# B&R Automation Studio project TD52 (part 48)

```iecst
	xMsg2303();

	OUT_CU.bMsg2303 :=	xMsg2303.Q;
	MM2VIS.bMsg2303 :=	xMsg2303.Q;

	(* W2415 mains import controller: Messsignalstörung Netzbezugs- Sollwert 	*)
	xMsg2415.Enable := bMsg2415_Enable AND IN_CU.tPB2MM.bParaSetupOk;
	xMsg2415.Set 	:= bMsg2415_Set;
	xMsg2415.PT 	:= T#1s;
	xMsg2415.Prio 	:= 4;
	xMsg2415.Reset 	:= FALSE;

	xMsg2415();

	OUT_CU.bMsg2415 :=	xMsg2415.Q;
	MM2VIS.bMsg2415 :=	xMsg2415.Q;

	(* W2416 mains import controller: Messsignalstörung Netzbezugs- Istwert	*)
//	Para.bP_Mns_AnaIn_Enable := NOT Para.bP_Mns_MMU_Enable	;						(*necessary, because bP_Mns_AnaIn_Enable is not a parameter on VIS anymore*)

	xMsg2416.Enable := bMsg2416_Enable AND IN_CU.tPB2MM.bParaSetupOk;
	xMsg2416.Set 	:= bMsg2416_Set;
//	NOT IN_CU.tP_Mns_AnaIn.GoodQual;
	xMsg2416.PT		:= T#1s;
	xMsg2416.Prio 	:= 4;
	xMsg2416.Reset 	:= FALSE;

	xMsg2416();

	OUT_CU.bMsg2416 :=	xMsg2416.Q;
	MM2VIS.bMsg2416 :=	xMsg2416.Q;

	(* W2417 mains export power limit: Warning, if NEGATIVE Mains Import (= power export to the grid) is exceeding (<) the allowed limit (-Limit value)  *)
	xMsg2417.Enable := bMsg2417_Enable AND IN_CU.tPB2MM.bParaSetupOk;
	xMsg2417.Set 	:= bMsg2417_Set;
	xMsg2417.PT 	:= T#1s;
	xMsg2417.Prio 	:= 4;
	xMsg2417.Reset 	:= FALSE;
	xMsg2417();

	OUT_CU.bMsg2417 :=	xMsg2417.Q;
	MM2VIS.bMsg2417 :=	xMsg2417.Q;

	(* W2418  mains import controller limit 2:  Warning if positive Mains Import (= power drawn from the grid) is exceeding (>) the allowed limit (+Limit value)*)
	xMsg2418.Enable := bMsg2418_Enable AND IN_CU.tPB2MM.bParaSetupOk;
	xMsg2418.Set 	:= bMsg2418_Set;
	xMsg2418.PT 	:= T#1s;
	xMsg2418.Prio 	:= 4;
	xMsg2418.Reset 	:= FALSE;

	xMsg2418();

	OUT_CU.bMsg2418 :=	xMsg2418.Q;
	MM2VIS.bMsg2418 :=	xMsg2418.Q;

	(* B2419 operating message mns import ctr: Engine Demand Off (ex.Warning W2419) *)
	TP_EngDSS_Mains_Off(IN := NOT(OUT_CU.bEngDSS_Mains), PT := T#11s);
	xMsg2419.Enable := 	Para.bCtr_Mns_Enable;
	xMsg2419.Set := 	TP_EngDSS_Mains_Off.Q;
	xMsg2419.PT := 		T#1s;
	xMsg2419.Prio := 	5;
	IF xMsg2419.Set THEN iReset_Msg2419 := iDelay_MsgAutoReset_100ms; ELSE iReset_Msg2419 := LIMIT(0, iReset_Msg2419 -1,32767); END_IF		(* activate 'Message Hold Time' to avoid log clathering by repeated OpMsg entries *)
	xMsg2419.Reset := 	iReset_Msg2419 < 1;		//.Reset := TRUE;
//
	xMsg2419();
//
	OUT_CU.bMsg2419 :=		xMsg2419.Q;	//  := TP_EngDSS_Mains_Off.Q;	//
	MM2VIS.bMsg2419 :=		xMsg2419.Q;	//	:= TP_EngDSS_Mains_Off.Q;	//

	(* B2420 operating message mns import ctr: Engine Demand On (ex. warning W2420)*)
	TP_EngDSS_Mains(IN := OUT_CU.bEngDSS_Mains, PT := T#11s);
	xMsg2420.Enable := 	Para.bCtr_Mns_Enable;
	xMsg2420.Set := 	TP_EngDSS_Mains.Q;
	xMsg2420.PT := 		T#1s;
	xMsg2420.Prio := 	5;

	IF xMsg2420.Set THEN iReset_Msg2420 := iDelay_MsgAutoReset_100ms; ELSE iReset_Msg2420 := LIMIT(0, iReset_Msg2420 -1,32767); END_IF		(* activate 'Message Hold Time' to avoid log clathering by repeated OpMsg entries *)
	xMsg2420.Reset := 	iReset_Msg2420 < 1;		//.Reset := TRUE;
//
	xMsg2420();
//
	OUT_CU.bMsg2420 :=		xMsg2420.Q;		// := TP_EngDSS_Mains.Q;		//
	MM2VIS.bMsg2420 :=		xMsg2420.Q;		// := TP_EngDSS_Mains.Q;		//

(*  Debug Info only (may be removed in tested versions)  *)
	bCtr_Mns_Options_2	:= Para.iCtr_Mns_Options.2;
	bCtr_Mns_Options_3	:= Para.iCtr_Mns_Options.3;
	bCtr_Mns_Options_4	:= Para.iCtr_Mns_Options.4;
	bCtr_Mns_Options_5	:= Para.iCtr_Mns_Options.5;
	bCtr_Mns_Options_6	:= Para.iCtr_Mns_Options.6;
	bCtr_Mns_Options_7	:= Para.iCtr_Mns_Options.7;
	bCtr_Mns_Options_8	:= Para.iCtr_Mns_Options.8;			bCtr_Mns_Options_1;	bCtr_Mns_Options_9;	bCtr_Mns_Options_0;
	R_TRIG_Options(CLK := (VIS2MM.tCtr_Mns_In.Tune_PI OR VIS2MM.tCtr_Mns_In.Tune_PID) AND VIS2MM.tCtr_Mns_In.Tune_quality>0);
	IF R_TRIG_Options.Q AND IN_CU.iIdx_OMSS=0 THEN Para.iCtr_Mns_Options := Para.iCtr_Mns_Options + BOOL_TO_INT(VIS2MM.tCtr_Mns_In.Tune_PI) * VIS2MM.tCtr_Mns_In.Tune_quality - BOOL_TO_INT(VIS2MM.tCtr_Mns_In.Tune_PID) * VIS2MM.tCtr_Mns_In.Tune_quality ; END_IF			(*Debug options*)

	(*********************************************************)

		(* W3565 Messsignalstörung Generator Leistungssollwert *)
		xMsg3565.Enable := 	(Para.rI_P_Set_ExtAI_NormScalMin >= 0.004);  (* if signal check is ok AND scaling parameter Min has to be set >4mA*) 	(*old V3.40: monitoring active, if parameter p_soll_i1 is setted to 4mA or higher *)
		xMsg3565.Set := 	NOT IN_CU.tP_Set_ExtAI_Norm.GoodQual;
		xMsg3565.PT := 		T#2s;
		xMsg3565.Prio := 	4;
		xMsg3565.Reset := 	FALSE;

		xMsg3565();

		MM2VIS.bMsg3565 :=	xMsg3565.Q;
		OUT_CU.bMsg3565 :=	xMsg3565.Q;

		(* W9285 Measuring signal failure external voltage setpoint *)
		MM2VIS.bMsg9285 :=	IN_CU.bMsg[9285];

		(* W9286 Measuring signal failure external speed setpoint (Isolated operation) *)
		xMsg9286.Enable := 	(Para.rI_N_Set_ExtAI_NormScalMin >= 0.004) AND IN_CU.tN_Set_ExtAI_Norm.Exist AND IN_CU.tPB2MM.bParaSetupOk;
		xMsg9286.Set := 	NOT IN_CU.tN_Set_ExtAI_Norm.GoodQual;
		xMsg9286.PT := 		T#1s;
		xMsg9286.Prio := 	4;
		xMsg9286.Reset := 	FALSE;

		xMsg9286();

		MM2VIS.bMsg9286 :=	xMsg9286.Q;
		OUT_CU.bMsg9286 :=	xMsg9286.Q;

		(* W9287 Failure external speed / voltage controller *)
		xMsg9287.Enable := 	IN_CU.tExtCtrOk.GoodQual AND IN_CU.tPB2MM.bParaSetupOk;
		xMsg9287.Set := 	NOT IN_CU.tExtCtrOk.Di;
		xMsg9287.PT := 		T#1s;
		xMsg9287.Prio := 	4;
		xMsg9287.Reset := 	FALSE;

		xMsg9287();

		MM2VIS.bMsg9287 :=	xMsg9287.Q;
		OUT_CU.bMsg9287 :=	xMsg9287.Q;

	(*----------------------------------------------------------------------------*)
	(* OPERATING MESSAGES: connect activation bits here customized 				  *)
	(*----------------------------------------------------------------------------*)

		OUT_CU.bMsg3232;// :=		FALSE;	(* B3232 reserve operating message 1 *)
		OUT_CU.bMsg3233;// :=		FALSE;	(* B3233 reserve operating message 2 *)
		OUT_CU.bMsg3234 ;// :=		FALSE;	(* B3234 reserve operating message 3 *)
		OUT_CU.bMsg3235 ;// :=		FALSE;	(* B3235 reserve operating message 4 *)
		OUT_CU.bMsg3236 ;// := 		FALSE;	(* B3236 reserve operating message 5 *)
		OUT_CU.bMsg3237 ;// := 		FALSE;	(* B3237 reserve operating message 6 *)

		OUT_CU.bMsg3250 ;// := 		FALSE;	(* B3250 reserve operating message 7 *)
		OUT_CU.bMsg3251 ;// := 		FALSE;	(* B3251 reserve operating message 8 *)

		OUT_CU.bMsg3601 ;// := 		FALSE;	(* B3601 reserve operating message 9 *)
		OUT_CU.bMsg3602 ;// := 		FALSE;	(* B3602 reserve operating message 10 *)
		OUT_CU.bMsg3603 ;// := 		FALSE;	(* B3603 reserve operating message 11 *)
		OUT_CU.bMsg3604 ;// := 		FALSE;	(* B3604 reserve operating message 12 *)
		OUT_CU.bMsg3605 ;// := 		FALSE;	(* B3605 reserve operating message 13 *)
		OUT_CU.bMsg3606 ;// := 		FALSE;	(* B3606 reserve operating message 14 *)
		OUT_CU.bMsg3607 ;// := 		FALSE;	(* B3607 reserve operating message 15 *)
		OUT_CU.bMsg3608 ;// := 		FALSE;	(* B3608 reserve operating message 16 *)
		OUT_CU.bMsg3609 ;// := 		FALSE;	(* B3609 reserve operating message 17 *)
		OUT_CU.bMsg3610 ;// := 		FALSE;	(* B3610 reserve operating message 18 *)

		OUT_CU.bMsg3611 ;// := 		FALSE;	(* B3611 reserve operating message 19 *)
		OUT_CU.bMsg3612 ;// := 		FALSE;	(*  	 reserve operating message 20 *)
		OUT_CU.bMsg3613 ;// := 		FALSE;	(* 		 reserve operating message 21 *)
		OUT_CU.bMsg3614 ;// := 		FALSE;	(* 		 reserve operating message 22 *)
		OUT_CU.bMsg3615 ;// := 		FALSE;	(* 		 reserve operating message 23 *)
		OUT_CU.bMsg3616 ;// := 		FALSE;	(* 		 reserve operating message 24 *)
		OUT_CU.bMsg3617 ;// := 		FALSE;	(* 		 reserve operating message 25 *)
		OUT_CU.bMsg3618 ;// := 		FALSE;	(* 		 reserve operating message 26 *)
		OUT_CU.bMsg3619 ;// := 		FALSE;	(* 		 reserve operating message 27 *)
		OUT_CU.bMsg3620 ;// := 		FALSE;	(* 		 reserve operating message 28 *)

		OUT_CU.bMsg3621 ;// := 		FALSE;	(* B3621 reserve operating message 29 *)
		OUT_CU.bMsg3622 ;// := 		FALSE;	(* 		 reserve operating message 30 *)
		OUT_CU.bMsg3623 ;// := 		FALSE;	(* 		 reserve operating message 31 *)
		OUT_CU.bMsg3624 ;// := 		FALSE;	(* 		 reserve operating message 32 *)
		OUT_CU.bMsg3625 ;// := 		FALSE;	(* 		 reserve operating message 33 *)
		OUT_CU.bMsg3626 ;// := 		FALSE;	(* 		 reserve operating message 34 *)
		OUT_CU.bMsg3627 ;// := 		FALSE;	(* 		 reserve operating message 35 *)
		OUT_CU.bMsg3628 ;// := 		FALSE;	(* 		 reserve operating message 36 *)
		OUT_CU.bMsg3629 ;// := 		FALSE;	(* 		 reserve operating message 37 *)
		OUT_CU.bMsg3630 ;// := 		FALSE;	(* 		 reserve operating message 38 *)

		OUT_CU.bMsg3631 ;// := 		FALSE;	(* 		 reserve operating message 39 *)
		OUT_CU.bMsg3632 ;// := 		FALSE;	(* 		 reserve operating message 40 *)
		OUT_CU.bMsg3633 ;// := 		FALSE;	(* 		 reserve operating message 41 *)
		OUT_CU.bMsg3634 ;// := 		FALSE;	(* 		 reserve operating message 42 *)
		OUT_CU.bMsg3635 ;// := 		FALSE;	(* 		 reserve operating message 43 *)
		OUT_CU.bMsg3636 ;// := 		FALSE;	(* 		 reserve operating message 44 *)
		OUT_CU.bMsg3637 ;// := 		FALSE;	(* 		 reserve operating message 45 *)
		OUT_CU.bMsg3638 ;// := 		FALSE;	(* 		 reserve operating message 46 *)
		OUT_CU.bMsg3639 ;// := 		FALSE;	(* 		 reserve operating message 47 *)
		OUT_CU.bMsg3640 ;// := 		FALSE;	(* 		 reserve operating message 48 *)

		OUT_CU.bMsg3641 ;// := 		FALSE;	(* B3641 reserve operating message 49 *)
		OUT_CU.bMsg3642 ;// := 		FALSE;	(* 		 reserve operating message 50 *)
		OUT_CU.bMsg3643 ;// := 		FALSE;	(* 		 reserve operating message 51 *)
		OUT_CU.bMsg3644 ;// := 		FALSE;	(* 		 reserve operating message 52 *)
		OUT_CU.bMsg3645 ;// := 		FALSE;	(* 		 reserve operating message 53 *)
		OUT_CU.bMsg3646 ;// := 		FALSE;	(* 		 reserve operating message 54 *)
		OUT_CU.bMsg3647 ;// := 		FALSE;	(* 		 reserve operating message 55 *)
		OUT_CU.bMsg3648 ;// := 		FALSE;	(* 		 reserve operating message 56 *)
		OUT_CU.bMsg3649 ;// := 		FALSE;	(* 		 reserve operating message 57 *)
		OUT_CU.bMsg3650 ;// := 		FALSE;	(* 		 reserve operating message 58 *)

		OUT_CU.bMsg3651 ;// := 		FALSE;	(* 		 reserve operating message 59 *)
		OUT_CU.bMsg3652 ;// := 		FALSE;	(* 		 reserve operating message 60 *)
		OUT_CU.bMsg3653 ;// := 		FALSE;	(* 		 reserve operating message 61 *)
		OUT_CU.bMsg3654 ;// := 		FALSE;	(* 		 reserve operating message 62 *)
		OUT_CU.bMsg3655 ;// := 		FALSE;	(* 		 reserve operating message 63 *)
		OUT_CU.bMsg3656 ;// := 		FALSE;	(* 		 reserve operating message 64 *)
		OUT_CU.bMsg3657 ;// := 		FALSE;	(* 		 reserve operating message 65 *)
		OUT_CU.bMsg3658 ;// := 		FALSE;	(* 		 reserve operating message 66 *)
		OUT_CU.bMsg3659 ;// := 		FALSE;	(* 		 reserve operating message 67 *)
		OUT_CU.bMsg3660 ;// := 		FALSE;	(* 		 reserve operating message 68 *)

		OUT_CU.bMsg3661 ;// := 		FALSE;	(* B3661 reserve operating message 69 *)
		OUT_CU.bMsg3662 ;// := 		FALSE;	(* 		 reserve operating message 70 *)
		OUT_CU.bMsg3663 ;// := 		FALSE;	(* 		 reserve operating message 71 *)
		OUT_CU.bMsg3664 ;// := 		FALSE;	(* 		 reserve operating message 72 *)
		OUT_CU.bMsg3665 ;// := 		FALSE;	(* 		 reserve operating message 73 *)
		OUT_CU.bMsg3666 ;// := 		FALSE;	(* 		 reserve operating message 74 *)
		OUT_CU.bMsg3667 ;// := 		FALSE;	(* 		 reserve operating message 75 *)
		OUT_CU.bMsg3668 ;// := 		FALSE;	(* 		 reserve operating message 76 *)
		OUT_CU.bMsg3669 ;// := 		FALSE;	(* 		 reserve operating message 77 *)
		OUT_CU.bMsg3670 ;// := 		FALSE;	(* 		 reserve operating message 78 *)

		OUT_CU.bMsg3671 ;// := 		FALSE;	(* 		 reserve operating message 79 *)
		OUT_CU.bMsg3672 ;// := 		FALSE;	(* 		 reserve operating message 80 *)
		OUT_CU.bMsg3673 ;// := 		FALSE;	(* 		 reserve operating message 81 *)
		OUT_CU.bMsg3674 ;// := 		FALSE;	(* 		 reserve operating message 82 *)
		OUT_CU.bMsg3675 ;// := 		FALSE;	(* 		 reserve operating message 83 *)
		OUT_CU.bMsg3676 ;// := 		FALSE;	(* 		 reserve operating message 84 *)
		OUT_CU.bMsg3677 ;// := 		FALSE;	(* 		 reserve operating message 85 *)
		OUT_CU.bMsg3678 ;// := 		FALSE;	(* 		 reserve operating message 86 *)
		OUT_CU.bMsg3679 ;// := 		FALSE;	(* 		 reserve operating message 87 *)
		OUT_CU.bMsg3680 ;// := 		FALSE;	(* 		 reserve operating message 88 *)

		OUT_CU.bMsg3681 ;// := 		FALSE;	(* B3681 reserve operating message 89 *)
		OUT_CU.bMsg3682 ;// := 		FALSE;	(* 		 reserve operating message 90 *)
		OUT_CU.bMsg3683 ;// := 		FALSE;	(* 		 reserve operating message 91 *)
		OUT_CU.bMsg3684 ;// := 		FALSE;	(* 		 reserve operating message 92 *)
		OUT_CU.bMsg3685 ;// := 		FALSE;	(* 		 reserve operating message 93 *)
		OUT_CU.bMsg3686 ;// := 		FALSE;	(* 		 reserve operating message 94 *)
		OUT_CU.bMsg3687 ;// := 		FALSE;	(* 		 reserve operating message 95 *)
		OUT_CU.bMsg3688 ;// := 		FALSE;	(* 		 reserve operating message 96 *)
		OUT_CU.bMsg3689 ;// := 		FALSE;	(* 		 reserve operating message 97 *)
		OUT_CU.bMsg3690 ;// := 		FALSE;	(* 		 reserve operating message 98 *)

		OUT_CU.bMsg3691 ;// := 		FALSE;	(* 		 reserve operating message 99 *)
		OUT_CU.bMsg3692 ;// := 		FALSE;	(* 		 reserve operating message 100 *)
		OUT_CU.bMsg3693 ;// := 		FALSE;	(* 		 reserve operating message 101 *)
		OUT_CU.bMsg3694 ;// := 		FALSE;	(* 		 reserve operating message 102 *)
		OUT_CU.bMsg3695 ;// := 		FALSE;	(* 		 reserve operating message 103 *)
		OUT_CU.bMsg3696 ;// := 		FALSE;	(* 		 reserve operating message 104 *)
		OUT_CU.bMsg3697 ;// := 		FALSE;	(* 		 reserve operating message 105 *)
		OUT_CU.bMsg3698 ;// := 		FALSE;	(* 		 reserve operating message 106 *)
		OUT_CU.bMsg3699 ;// := 		FALSE;	(* 		 reserve operating message 107 *)
		OUT_CU.bMsg3700 ;// := 		FALSE;	(* 		 reserve operating message 108 *)

		OUT_CU.bMsg6701 ;// := 		FALSE;	(* B6701 reserve operating message 109 *) (*import HMI Extension *)
		OUT_CU.bMsg6702 ;// := 		FALSE;	(* B6702 reserve operating message 110 *) (*import HMI Extension *)
		OUT_CU.bMsg6703 ;// := 		FALSE;	(* B6703 reserve operating message 111 *) (*import HMI Extension *)
		OUT_CU.bMsg6704 ;// := 		FALSE;	(* B6704 reserve operating message 112 *) (*import HMI Extension *)
		OUT_CU.bMsg6705 ;// := 		FALSE;	(* B6705 reserve operating message 113 *) (*import HMI Extension *)
		OUT_CU.bMsg6706 ;// := 		FALSE;	(* B6706 reserve operating message 114 *) (*import HMI Extension *)
		OUT_CU.bMsg6707 ;// := 		FALSE;	(* B6707 reserve operating message 115 *) (*import HMI Extension *)
		OUT_CU.bMsg6708 ;// := 		FALSE;	(* B6708 reserve operating message 116 *) (*import HMI Extension *)
		OUT_CU.bMsg6709 ;// := 		FALSE;	(* B6709 reserve operating message 117 *) (*import HMI Extension *)
		OUT_CU.bMsg6710 ;// := 		FALSE;	(* B6710 reserve operating message 118 *) (*import HMI Extension *)

		OUT_CU.bMsg6711 ;// := 		FALSE;	(* B6711 reserve operating message 119 *) (*import HMI Extension *)
		OUT_CU.bMsg6712 ;// := 		FALSE;	(* B6712 reserve operating message 120 *) (*import HMI Extension *)
		OUT_CU.bMsg6713 ;// := 		FALSE;	(* B6713 reserve operating message 121 *) (*import HMI Extension *)
		OUT_CU.bMsg6714 ;// := 		FALSE;	(* B6714 reserve operating message 122 *) (*import HMI Extension *)
		OUT_CU.bMsg6715 ;// := 		FALSE;	(* B6715 reserve operating message 123 *) (*import HMI Extension *)
		OUT_CU.bMsg6716 ;// := 		FALSE;	(* B6716 reserve operating message 124 *) (*import HMI Extension *)
		OUT_CU.bMsg6717 ;// := 		FALSE;	(* B6717 reserve operating message 125 *) (*import HMI Extension *)
		OUT_CU.bMsg6718 ;// := 		FALSE;	(* B6718 reserve operating message 126 *) (*import HMI Extension *)
		OUT_CU.bMsg6719 ;// := 		FALSE;	(* B6719 reserve operating message 127 *) (*import HMI Extension *)
		OUT_CU.bMsg6720 ;// := 		FALSE;	(* B6720 reserve operating message 128 *) (*import HMI Extension *)

		OUT_CU.bMsg6721 ;// := 		FALSE;	(* B6721 reserve operating message 129 *) (*import HMI Extension *)
		OUT_CU.bMsg6722 ;// := 		FALSE;	(* B6722 reserve operating message 130 *) (*import HMI Extension *)
		OUT_CU.bMsg6723 ;// := 		FALSE;	(* B6723 reserve operating message 131 *) (*import HMI Extension *)
		OUT_CU.bMsg6724 ;// := 		FALSE;	(* B6724 reserve operating message 132 *) (*import HMI Extension *)
		OUT_CU.bMsg6725 ;// := 		FALSE;	(* B6725 reserve operating message 133 *) (*import HMI Extension *)
		OUT_CU.bMsg6726 ;// := 		FALSE;	(* B6726 reserve operating message 134 *) (*import HMI Extension *)
		OUT_CU.bMsg6727 ;// := 		FALSE;	(* B6727 reserve operating message 135 *) (*import HMI Extension *)
		OUT_CU.bMsg6728 ;// := 		FALSE;	(* B6728 reserve operating message 136 *) (*import HMI Extension *)
		OUT_CU.bMsg6729 ;// := 		FALSE;	(* B6729 reserve operating message 137 *) (*import HMI Extension *)
		OUT_CU.bMsg6730 ;// := 		FALSE;	(* B6730 reserve operating message 138 *) (*import HMI Extension *)

		OUT_CU.bMsg6731 ;// := 		FALSE;	(* B6731 reserve operating message 139 *) (*import HMI Extension *)
		OUT_CU.bMsg6732 ;// := 		FALSE;	(* B6732 reserve operating message 140 *) (*import HMI Extension *)
		OUT_CU.bMsg6733 ;// := 		FALSE;	(* B6733 reserve operating message 141 *) (*import HMI Extension *)
		OUT_CU.bMsg6734 ;// := 		FALSE;	(* B6734 reserve operating message 142 *) (*import HMI Extension *)
		OUT_CU.bMsg6735 ;// := 		FALSE;	(* B6735 reserve operating message 143 *) (*import HMI Extension *)
		OUT_CU.bMsg6736 ;// := 		FALSE;	(* B6736 reserve operating message 144 *) (*import HMI Extension *)
		OUT_CU.bMsg6737 ;// := 		FALSE;	(* B6737 reserve operating message 145 *) (*import HMI Extension *)
		OUT_CU.bMsg6738 ;// := 		FALSE;	(* B6738 reserve operating message 146 *) (*import HMI Extension *)
		OUT_CU.bMsg6739 ;// := 		FALSE;	(* B6739 reserve operating message 147 *) (*import HMI Extension *)
		OUT_CU.bMsg6740 ;// := 		FALSE;	(* B6740 reserve operating message 148 *) (*import HMI Extension *)

		OUT_CU.bMsg6741 ;// := 		FALSE;	(* B6741 reserve operating message 149 *) (*import HMI Extension *)
		OUT_CU.bMsg6742 ;// := 		FALSE;	(* B6742 reserve operating message 150 *) (*import HMI Extension *)
		OUT_CU.bMsg6743 ;// := 		FALSE;	(* B6743 reserve operating message 151 *) (*import HMI Extension *)
		OUT_CU.bMsg6744 ;// := 		FALSE;	(* B6744 reserve operating message 152 *) (*import HMI Extension *)
		OUT_CU.bMsg6745 ;// := 		FALSE;	(* B6745 reserve operating message 153 *) (*import HMI Extension *)
		OUT_CU.bMsg6746 ;// := 		FALSE;	(* B6746 reserve operating message 154 *) (*import HMI Extension *)
		OUT_CU.bMsg6747 ;// := 		FALSE;	(* B6747 reserve operating message 155 *) (*import HMI Extension *)
		OUT_CU.bMsg6748 ;// := 		FALSE;	(* B6748 reserve operating message 156 *) (*import HMI Extension *)
		OUT_CU.bMsg6749 ;// := 		FALSE;	(* B6749 reserve operating message 157 *) (*import HMI Extension *)
		OUT_CU.bMsg6750 ;// := 		FALSE;	(* B6750 reserve operating message 158 *) (*import HMI Extension *)

		OUT_CU.bMsg6751 ;// := 		FALSE;	(* B6751 reserve operating message 159 *) (*import HMI Extension *)
		OUT_CU.bMsg6752 ;// := 		FALSE;	(* B6752 reserve operating message 160 *) (*import HMI Extension *)
		OUT_CU.bMsg6753 ;// := 		FALSE;	(* B6753 reserve operating message 161 *) (*import HMI Extension *)
		OUT_CU.bMsg6754 ;// := 		FALSE;	(* B6754 reserve operating message 162 *) (*import HMI Extension *)
		OUT_CU.bMsg6755 ;// := 		FALSE;	(* B6755 reserve operating message 163 *) (*import HMI Extension *)
		OUT_CU.bMsg6756 ;// := 		FALSE;	(* B6756 reserve operating message 164 *) (*import HMI Extension *)
		OUT_CU.bMsg6757 ;// := 		FALSE;	(* B6757 reserve operating message 165 *) (*import HMI Extension *)
		OUT_CU.bMsg6758 ;// := 		FALSE;	(* B6758 reserve operating message 166 *) (*import HMI Extension *)
		OUT_CU.bMsg6759 ;// := 		FALSE;	(* B6759 reserve operating message 167 *) (*import HMI Extension *)
		OUT_CU.bMsg6760 ;// := 		FALSE;	(* B6760 reserve operating message 168 *) (*import HMI Extension *)

		OUT_CU.bMsg6761 ;// := 		FALSE;	(* B6761 reserve operating message 169 *) (*import HMI Extension *)
		OUT_CU.bMsg6762 ;// := 		FALSE;	(* B6762 reserve operating message 170 *) (*import HMI Extension *)
		OUT_CU.bMsg6763 ;// := 		FALSE;	(* B6763 reserve operating message 171 *) (*import HMI Extension *)
		OUT_CU.bMsg6764 ;// := 		FALSE;	(* B6764 reserve operating message 172 *) (*import HMI Extension *)
		OUT_CU.bMsg6765 ;// := 		FALSE;	(* B6765 reserve operating message 173 *) (*import HMI Extension *)
		OUT_CU.bMsg6766 ;// := 		FALSE;	(* B6766 reserve operating message 174 *) (*import HMI Extension *)
		OUT_CU.bMsg6767 ;// := 		FALSE;	(* B6767 reserve operating message 175 *) (*import HMI Extension *)
		OUT_CU.bMsg6768 ;// := 		FALSE;	(* B6768 reserve operating message 176 *) (*import HMI Extension *)
		OUT_CU.bMsg6769 ;// := 		FALSE;	(* B6769 reserve operating message 177 *) (*import HMI Extension *)
		OUT_CU.bMsg6770 ;// := 		FALSE;	(* B6770 reserve operating message 178 *) (*import HMI Extension *)

		OUT_CU.bMsg6771 ;// := 		FALSE;	(* B6771 reserve operating message 179 *) (*import HMI Extension *)
		OUT_CU.bMsg6772 ;// := 		FALSE;	(* B6772 reserve operating message 180 *) (*import HMI Extension *)
		OUT_CU.bMsg6773 ;// := 		FALSE;	(* B6773 reserve operating message 181 *) (*import HMI Extension *)
		OUT_CU.bMsg6774 ;// := 		FALSE;	(* B6774 reserve operating message 182 *) (*import HMI Extension *)
		OUT_CU.bMsg6775 ;// := 		FALSE;	(* B6775 reserve operating message 183 *) (*import HMI Extension *)
		OUT_CU.bMsg6776 ;// := 		FALSE;	(* B6776 reserve operating message 184 *) (*import HMI Extension *)
		OUT_CU.bMsg6777 ;// := 		FALSE;	(* B6777 reserve operating message 185 *) (*import HMI Extension *)
		OUT_CU.bMsg6778 ;// := 		FALSE;	(* B6778 reserve operating message 186 *) (*import HMI Extension *)
		OUT_CU.bMsg6779 ;// := 		FALSE;	(* B6779 reserve operating message 187 *) (*import HMI Extension *)
		OUT_CU.bMsg6780 ;// := 		FALSE;	(* B6780 reserve operating message 188 *) (*import HMI Extension *)

		OUT_CU.bMsg6781 ;// := 		FALSE;	(* B6781 reserve operating message 189 *) (*import HMI Extension *)
		OUT_CU.bMsg6782 ;// := 		FALSE;	(* B6782 reserve operating message 190 *) (*import HMI Extension *)
		OUT_CU.bMsg6783 ;// := 		FALSE;	(* B6783 reserve operating message 191 *) (*import HMI Extension *)
		OUT_CU.bMsg6784 ;// := 		FALSE;	(* B6784 reserve operating message 192 *) (*import HMI Extension *)
		OUT_CU.bMsg6785 ;// := 		FALSE;	(* B6785 reserve operating message 193 *) (*import HMI Extension *)
		OUT_CU.bMsg6786 ;// := 		FALSE;	(* B6786 reserve operating message 194 *) (*import HMI Extension *)
		OUT_CU.bMsg6787 ;// := 		FALSE;	(* B6787 reserve operating message 195 *) (*import HMI Extension *)
		OUT_CU.bMsg6788 ;// := 		FALSE;	(* B6788 reserve operating message 196 *) (*import HMI Extension *)
		OUT_CU.bMsg6789 ;// := 		FALSE;	(* B6789 reserve operating message 197 *) (*import HMI Extension *)
		OUT_CU.bMsg6790 ;// := 		FALSE;	(* B6790 reserve operating message 198 *) (*import HMI Extension *)

		OUT_CU.bMsg6791 ;// := 		FALSE;	(* B6791 reserve operating message 199 *) (*import HMI Extension *)
		OUT_CU.bMsg6792 ;// := 		FALSE;	(* B6792 reserve operating message 200 *) (*import HMI Extension *)
		OUT_CU.bMsg6793 ;// := 		FALSE;	(* B6793 reserve operating message 201 *) (*import HMI Extension *)
		OUT_CU.bMsg6794 ;// := 		FALSE;	(* B6794 reserve operating message 202 *) (*import HMI Extension *)
		OUT_CU.bMsg6795 ;// := 		FALSE;	(* B6795 reserve operating message 203 *) (*import HMI Extension *)
		OUT_CU.bMsg6796 ;// := 		FALSE;	(* B6796 reserve operating message 204 *) (*import HMI Extension *)
		OUT_CU.bMsg6797 ;// := 		FALSE;	(* B6797 reserve operating message 205 *) (*import HMI Extension *)
		OUT_CU.bMsg6798 ;// := 		FALSE;	(* B6798 reserve operating message 206 *) (*import HMI Extension *)
		OUT_CU.bMsg6799 ;// := 		FALSE;	(* B6799 reserve operating message 207 *) (*import HMI Extension *)
		OUT_CU.bMsg6800 ;// := 		FALSE;	(* B6800 reserve operating message 208 *) (*import HMI Extension *)

		OUT_CU.bMsg6801 ;// := 		FALSE;	(* B6801 reserve operating message 209 *) (*import HMI Extension *)
		OUT_CU.bMsg6802 ;// := 		FALSE;	(* B6802 reserve operating message 210 *) (*import HMI Extension *)
		OUT_CU.bMsg6803 ;// := 		FALSE;	(* B6803 reserve operating message 211 *) (*import HMI Extension *)
		OUT_CU.bMsg6804 ;// := 		FALSE;	(* B6804 reserve operating message 212 *) (*import HMI Extension *)
		OUT_CU.bMsg6805 ;// := 		FALSE;	(* B6805 reserve operating message 213 *) (*import HMI Extension *)
		OUT_CU.bMsg6806 ;// := 		FALSE;	(* B6806 reserve operating message 214 *) (*import HMI Extension *)
		OUT_CU.bMsg6807 ;// := 		FALSE;	(* B6807 reserve operating message 215 *) (*import HMI Extension *)
		OUT_CU.bMsg6808 ;// := 		FALSE;	(* B6808 reserve operating message 216 *) (*import HMI Extension *)
		OUT_CU.bMsg6809 ;// := 		FALSE;	(* B6809 reserve operating message 217 *) (*import HMI Extension *)
		OUT_CU.bMsg6810 ;// := 		FALSE;	(* B6810 reserve operating message 218 *) (*import HMI Extension *)

		OUT_CU.bMsg6811 ;// := 		FALSE;	(* B6811 reserve operating message 219 *) (*import HMI Extension *)
		OUT_CU.bMsg6812 ;// := 		FALSE;	(* B6812 reserve operating message 220 *) (*import HMI Extension *)
		OUT_CU.bMsg6813 ;// := 		FALSE;	(* B6813 reserve operating message 221 *) (*import HMI Extension *)
		OUT_CU.bMsg6814 ;// := 		FALSE;	(* B6814 reserve operating message 222 *) (*import HMI Extension *)
		OUT_CU.bMsg6815 ;// := 		FALSE;	(* B6815 reserve operating message 223 *) (*import HMI Extension *)
		OUT_CU.bMsg6816 ;// := 		FALSE;	(* B6816 reserve operating message 224 *) (*import HMI Extension *)
		OUT_CU.bMsg6817 ;// := 		FALSE;	(* B6817 reserve operating message 225 *) (*import HMI Extension *)
		OUT_CU.bMsg6818 ;// := 		FALSE;	(* B6818 reserve operating message 226 *) (*import HMI Extension *)
		OUT_CU.bMsg6819 ;// := 		FALSE;	(* B6819 reserve operating message 227 *) (*import HMI Extension *)
		OUT_CU.bMsg6820 ;// := 		FALSE;	(* B6820 reserve operating message 228 *) (*import HMI Extension *)

		OUT_CU.bMsg6821 ;// := 		FALSE;	(* B6821 reserve operating message 229 *) (*import HMI Extension *)
		OUT_CU.bMsg6822 ;// := 		FALSE;	(* B6822 reserve operating message 230 *) (*import HMI Extension *)
		OUT_CU.bMsg6823 ;// := 		FALSE;	(* B6823 reserve operating message 231 *) (*import HMI Extension *)
		OUT_CU.bMsg6824 ;// := 		FALSE;	(* B6824 reserve operating message 232 *) (*import HMI Extension *)
		OUT_CU.bMsg6825 ;// := 		FALSE;	(* B6825 reserve operating message 233 *) (*import HMI Extension *)
		OUT_CU.bMsg6826 ;// := 		FALSE;	(* B6826 reserve operating message 234 *) (*import HMI Extension *)
		OUT_CU.bMsg6827 ;// := 		FALSE;	(* B6827 reserve operating message 235 *) (*import HMI Extension *)
		OUT_CU.bMsg6828 ;// := 		FALSE;	(* B6828 reserve operating message 236 *) (*import HMI Extension *)
		OUT_CU.bMsg6829 ;// := 		FALSE;	(* B6829 reserve operating message 237 *) (*import HMI Extension *)
		OUT_CU.bMsg6830 ;// := 		FALSE;	(* B6830 reserve operating message 238 *) (*import HMI Extension *)

		OUT_CU.bMsg6831 ;// := 		FALSE;	(* B6831 reserve operating message 239 *) (*import HMI Extension *)
		OUT_CU.bMsg6832 ;// := 		FALSE;	(* B6832 reserve operating message 240 *) (*import HMI Extension *)
		OUT_CU.bMsg6833 ;// := 		FALSE;	(* B6833 reserve operating message 241 *) (*import HMI Extension *)
		OUT_CU.bMsg6834 ;// := 		FALSE;	(* B6834 reserve operating message 242 *) (*import HMI Extension *)
		OUT_CU.bMsg6835 ;// := 		FALSE;	(* B6835 reserve operating message 243 *) (*import HMI Extension *)
		OUT_CU.bMsg6836 ;// := 		FALSE;	(* B6836 reserve operating message 244 *) (*import HMI Extension *)
		OUT_CU.bMsg6837 ;// := 		FALSE;	(* B6837 reserve operating message 245 *) (*import HMI Extension *)
		OUT_CU.bMsg6838 ;// := 		FALSE;	(* B6838 reserve operating message 246 *) (*import HMI Extension *)
		OUT_CU.bMsg6839 ;// := 		FALSE;	(* B6839 reserve operating message 247 *) (*import HMI Extension *)
		OUT_CU.bMsg6840 ;// := 		FALSE;	(* B6840 reserve operating message 248 *) (*import HMI Extension *)

		OUT_CU.bMsg6841 ;// := 		FALSE;	(* B6841 reserve operating message 249 *) (*import HMI Extension *)
		OUT_CU.bMsg6842 ;// := 		FALSE;	(* B6842 reserve operating message 250 *) (*import HMI Extension *)
		OUT_CU.bMsg6843 ;// := 		FALSE;	(* B6843 reserve operating message 251 *) (*import HMI Extension *)
		OUT_CU.bMsg6844 ;// := 		FALSE;	(* B6844 reserve operating message 252 *) (*import HMI Extension *)
		OUT_CU.bMsg6845 ;// := 		FALSE;	(* B6845 reserve operating message 253 *) (*import HMI Extension *)
		OUT_CU.bMsg6846 ;// := 		FALSE;	(* B6846 reserve operating message 254 *) (*import HMI Extension *)
		OUT_CU.bMsg6847 ;// := 		FALSE;	(* B6847 reserve operating message 255 *) (*import HMI Extension *)
		OUT_CU.bMsg6848 ;// := 		FALSE;	(* B6848 reserve operating message 256 *) (*import HMI Extension *)
		OUT_CU.bMsg6849 ;// := 		FALSE;	(* B6849 reserve operating message 257 *) (*import HMI Extension *)
		OUT_CU.bMsg6850 ;// := 		FALSE;	(* B6850 reserve operating message 258 *) (*import HMI Extension *)

		OUT_CU.bMsg6851 ;// := 		FALSE;	(* B6851 reserve operating message 259 *) (*import HMI Extension *)
		OUT_CU.bMsg6852 ;// := 		FALSE;	(* B6852 reserve operating message 260 *) (*import HMI Extension *)
		OUT_CU.bMsg6853 ;// := 		FALSE;	(* B6853 reserve operating message 261 *) (*import HMI Extension *)
		OUT_CU.bMsg6854 ;// := 		FALSE;	(* B6854 reserve operating message 262 *) (*import HMI Extension *)
		OUT_CU.bMsg6855 ;// := 		FALSE;	(* B6855 reserve operating message 263 *) (*import HMI Extension *)
		OUT_CU.bMsg6856 ;// := 		FALSE;	(* B6856 reserve operating message 264 *) (*import HMI Extension *)
		OUT_CU.bMsg6857 ;// := 		FALSE;	(* B6857 reserve operating message 265 *) (*import HMI Extension *)
		OUT_CU.bMsg6858 ;// := 		FALSE;	(* B6858 reserve operating message 266 *) (*import HMI Extension *)
		OUT_CU.bMsg6859 ;// := 		FALSE;	(* B6859 reserve operating message 267 *) (*import HMI Extension *)
		OUT_CU.bMsg6860 ;// := 		FALSE;	(* B6860 reserve operating message 268 *) (*import HMI Extension *)

		OUT_CU.bMsg6861 ;// := 		FALSE;	(* B6861 reserve operating message 269 *) (*import HMI Extension *)
		OUT_CU.bMsg6862 ;// := 		FALSE;	(* B6862 reserve operating message 270 *) (*import HMI Extension *)
		OUT_CU.bMsg6863 ;// := 		FALSE;	(* B6863 reserve operating message 271 *) (*import HMI Extension *)
		OUT_CU.bMsg6864 ;// := 		FALSE;	(* B6864 reserve operating message 272 *) (*import HMI Extension *)
		OUT_CU.bMsg6865 ;// := 		FALSE;	(* B6865 reserve operating message 273 *) (*import HMI Extension *)
		OUT_CU.bMsg6866 ;// := 		FALSE;	(* B6866 reserve operating message 274 *) (*import HMI Extension *)
		OUT_CU.bMsg6867 ;// := 		FALSE;	(* B6867 reserve operating message 275 *) (*import HMI Extension *)
		OUT_CU.bMsg6868 ;// := 		FALSE;	(* B6868 reserve operating message 276 *) (*import HMI Extension *)
		OUT_CU.bMsg6869 ;// := 		FALSE;	(* B6869 reserve operating message 277 *) (*import HMI Extension *)
		OUT_CU.bMsg6870 ;// := 		FALSE;	(* B6870 reserve operating message 278 *) (*import HMI Extension *)

		OUT_CU.bMsg6871 ;// := 		FALSE;	(* B6871 reserve operating message 279 *) (*import HMI Extension *)
		OUT_CU.bMsg6872 ;// := 		FALSE;	(* B6872 reserve operating message 280 *) (*import HMI Extension *)
		OUT_CU.bMsg6873 ;// := 		FALSE;	(* B6873 reserve operating message 281 *) (*import HMI Extension *)
		OUT_CU.bMsg6874 ;// := 		FALSE;	(* B6874 reserve operating message 282 *) (*import HMI Extension *)
		OUT_CU.bMsg6875 ;// := 		FALSE;	(* B6875 reserve operating message 283 *) (*import HMI Extension *)
		OUT_CU.bMsg6876 ;// := 		FALSE;	(* B6876 reserve operating message 284 *) (*import HMI Extension *)
		OUT_CU.bMsg6877 ;// := 		FALSE;	(* B6877 reserve operating message 285 *) (*import HMI Extension *)
		OUT_CU.bMsg6878 ;// := 		FALSE;	(* B6878 reserve operating message 286 *) (*import HMI Extension *)
		OUT_CU.bMsg6879 ;// := 		FALSE;	(* B6879 reserve operating message 287 *) (*import HMI Extension *)
		OUT_CU.bMsg6880 ;// := 		FALSE;	(* B6880 reserve operating message 288 *) (*import HMI Extension *)

		OUT_CU.bMsg6881 ;// := 		FALSE;	(* B6881 reserve operating message 289 *) (*import HMI Extension *)
		OUT_CU.bMsg6882 ;// := 		FALSE;	(* B6882 reserve operating message 290 *) (*import HMI Extension *)
		OUT_CU.bMsg6883 ;// := 		FALSE;	(* B6883 reserve operating message 291 *) (*import HMI Extension *)
		OUT_CU.bMsg6884 ;// := 		FALSE;	(* B6884 reserve operating message 292 *) (*import HMI Extension *)
		OUT_CU.bMsg6885 ;// := 		FALSE;	(* B6885 reserve operating message 293 *) (*import HMI Extension *)
		OUT_CU.bMsg6886 ;// := 		FALSE;	(* B6886 reserve operating message 294 *) (*import HMI Extension *)
		OUT_CU.bMsg6887 ;// := 		FALSE;	(* B6887 reserve operating message 295 *) (*import HMI Extension *)
		OUT_CU.bMsg6888 ;// := 		FALSE;	(* B6888 reserve operating message 296 *) (*import HMI Extension *)
		OUT_CU.bMsg6889 ;// := 		FALSE;	(* B6889 reserve operating message 297 *) (*import HMI Extension *)
		OUT_CU.bMsg6890 ;// := 		FALSE;	(* B6890 reserve operating message 298 *) (*import HMI Extension *)

		OUT_CU.bMsg6891 ;// := 		FALSE;	(* B6891 reserve operating message 299 *) (*import HMI Extension *)
		OUT_CU.bMsg6892 ;// := 		FALSE;	(* B6892 reserve operating message 300 *) (*import HMI Extension *)
		OUT_CU.bMsg6893 ;// := 		FALSE;	(* B6893 reserve operating message 301 *) (*import HMI Extension *)
		OUT_CU.bMsg6894 ;// := 		FALSE;	(* B6894 reserve operating message 302 *) (*import HMI Extension *)
		OUT_CU.bMsg6895 ;// := 		FALSE;	(* B6895 reserve operating message 303 *) (*import HMI Extension *)
		OUT_CU.bMsg6896 ;// := 		FALSE;	(* B6896 reserve operating message 304 *) (*import HMI Extension *)
		OUT_CU.bMsg6897 ;// := 		FALSE;	(* B6897 reserve operating message 305 *) (*import HMI Extension *)
		OUT_CU.bMsg6898 ;// := 		FALSE;	(* B6898 reserve operating message 306 *) (*import HMI Extension *)
		OUT_CU.bMsg6899 ;// := 		FALSE;	(* B6899 reserve operating message 307 *) (*import HMI Extension *)
//OLD do not use		OUT_CU.bMsg8700 ;// := 		FALSE;	(* B4200 reserve operating message 308 *) (*import HMI Extension *)

	(*----------------------------------------------------------------------------*)
	(* NO CHANGES BEYOND THIS LINE necessary  *)
	(*----------------------------------------------------------------------------*)
	(*---------------------------------------------------------------------------*)
	(* general alarms for further module operations *)
	bGnlTrip1 := 		OUT_CU.tCU2AB.bGnlTrip1   OR IN_CU.tAB2CU.bGnlTrip1;
	bGnlTrip2 := 		OUT_CU.tCU2AB.bGnlTrip2   OR IN_CU.tAB2CU.bGnlTrip2;
	bGnlTrip3 := 		OUT_CU.tCU2AB.bGnlTrip3   OR IN_CU.tAB2CU.bGnlTrip3;
	bGnlWarning:=		OUT_CU.tCU2AB.bGnlWarning OR IN_CU.tAB2CU.bGnlWarning;

	bGnlTrip := 		bGnlTrip1 OR bGnlTrip2 OR bGnlTrip3;

	(*----------------------------------------------------------------------------*)
	(* MODULE OUTPUT INFO:  *)

//	OUT_CU.iCount1 := 		FALSE;	(* customized counter 1: ... *)
//	OUT_CU.iCount2 := 		FALSE;	(* customized counter 2: ... *)
//	OUT_CU.iCount3 := 		FALSE;	(* customized counter 3: ... *)
//	OUT_CU.iCount4 := 		FALSE;	(* customized counter 4: ... *)
//	(*...*)
//	OUT_CU.iCount19 := 		FALSE;	(* customized counter 19: ... *)
//	OUT_CU.iCount20 := 		FALSE;	(* customized counter 20: ... *)

	(*----------------------------------------------------------------------------*)

	(* Forwarding of spare alarm messages: *)
(*	MM2VIS.bMsg1601 :=	xMsg16[01].Q; *)		OUT_CU.bMsg1601 :=	xMsg16[01].Q;    (*remove duplicate MM2VIS handling*)
												OUT_CU.bMsg1602 :=	xMsg16[02].Q;    (*remove duplicate MM2VIS handling*)
												OUT_CU.bMsg1603 :=	xMsg16[03].Q;    (*remove duplicate MM2VIS handling*)
												OUT_CU.bMsg1604 :=	xMsg16[04].Q;		//ToDo..
												OUT_CU.bMsg1605 :=	xMsg16[05].Q;
												OUT_CU.bMsg1606 :=	xMsg16[06].Q;
												OUT_CU.bMsg1607 :=	xMsg16[07].Q;
												OUT_CU.bMsg1608 :=	xMsg16[08].Q;
												OUT_CU.bMsg1609 :=	xMsg16[09].Q;
												OUT_CU.bMsg1610 :=	xMsg16[10].Q;

	MM2VIS.bMsg1611 :=	xMsg16[11].Q;			OUT_CU.bMsg1611 :=	xMsg16[11].Q;
	MM2VIS.bMsg1612 :=	xMsg16[12].Q;			OUT_CU.bMsg1612 :=	xMsg16[12].Q;
	MM2VIS.bMsg1613 :=	xMsg16[13].Q;			OUT_CU.bMsg1613 :=	xMsg16[13].Q;
	MM2VIS.bMsg1614 :=	xMsg16[14].Q;			OUT_CU.bMsg1614 :=	xMsg16[14].Q;
	MM2VIS.bMsg1615 :=	xMsg16[15].Q;			OUT_CU.bMsg1615 :=	xMsg16[15].Q;
	MM2VIS.bMsg1616 :=	xMsg16[16].Q;			OUT_CU.bMsg1616 :=	xMsg16[16].Q;
	MM2VIS.bMsg1617 :=	xMsg16[17].Q;			OUT_CU.bMsg1617 :=	xMsg16[17].Q;
	MM2VIS.bMsg1618 :=	xMsg16[18].Q;			OUT_CU.bMsg1618 :=	xMsg16[18].Q;
	MM2VIS.bMsg1619 :=	xMsg16[19].Q;			OUT_CU.bMsg1619 :=	xMsg16[19].Q;
	MM2VIS.bMsg1620 :=	xMsg16[20].Q;			OUT_CU.bMsg1620 :=	xMsg16[20].Q;

	MM2VIS.bMsg1621 :=	xMsg16[21].Q;			OUT_CU.bMsg1621 :=	xMsg16[21].Q;
	MM2VIS.bMsg1622 :=	xMsg16[22].Q;			OUT_CU.bMsg1622 :=	xMsg16[22].Q;
	MM2VIS.bMsg1623 :=	xMsg16[23].Q;			OUT_CU.bMsg1623 :=	xMsg16[23].Q;
	MM2VIS.bMsg1624 :=	xMsg16[24].Q;			OUT_CU.bMsg1624 :=	xMsg16[24].Q;
	MM2VIS.bMsg1625 :=	xMsg16[25].Q;			OUT_CU.bMsg1625 :=	xMsg16[25].Q;
	MM2VIS.bMsg1626 :=	xMsg16[26].Q;			OUT_CU.bMsg1626 :=	xMsg16[26].Q;
	MM2VIS.bMsg1627 :=	xMsg16[27].Q;			OUT_CU.bMsg1627 :=	xMsg16[27].Q;
	MM2VIS.bMsg1628 :=	xMsg16[28].Q;			OUT_CU.bMsg1628 :=	xMsg16[28].Q;
	MM2VIS.bMsg1629 :=	xMsg16[29].Q;			OUT_CU.bMsg1629 :=	xMsg16[29].Q;
	MM2VIS.bMsg1630 :=	xMsg16[30].Q;			OUT_CU.bMsg1630 :=	xMsg16[30].Q;

	MM2VIS.bMsg1631 :=	xMsg16[31].Q;			OUT_CU.bMsg1631 :=	xMsg16[31].Q;
	MM2VIS.bMsg1632 :=	xMsg16[32].Q;			OUT_CU.bMsg1632 :=	xMsg16[32].Q;
	MM2VIS.bMsg1633 :=	xMsg16[33].Q;			OUT_CU.bMsg1633 :=	xMsg16[33].Q;
	MM2VIS.bMsg1634 :=	xMsg16[34].Q;			OUT_CU.bMsg1634 :=	xMsg16[34].Q;
	MM2VIS.bMsg1635 :=	xMsg16[35].Q;			OUT_CU.bMsg1635 :=	xMsg16[35].Q;
	MM2VIS.bMsg1636 :=	xMsg16[36].Q;			OUT_CU.bMsg1636 :=	xMsg16[36].Q;
	MM2VIS.bMsg1637 :=	xMsg16[37].Q;			OUT_CU.bMsg1637 :=	xMsg16[37].Q;
	MM2VIS.bMsg1638 :=	xMsg16[38].Q;			OUT_CU.bMsg1638 :=	xMsg16[38].Q;
	MM2VIS.bMsg1639 :=	xMsg16[39].Q;			OUT_CU.bMsg1639 :=	xMsg16[39].Q;
	MM2VIS.bMsg1640 :=	xMsg16[40].Q;			OUT_CU.bMsg1640 :=	xMsg16[40].Q;

	MM2VIS.bMsg1641 :=	xMsg16[41].Q;			OUT_CU.bMsg1641 :=	xMsg16[41].Q;
	MM2VIS.bMsg1642 :=	xMsg16[42].Q;			OUT_CU.bMsg1642 :=	xMsg16[42].Q;
	MM2VIS.bMsg1643 :=	xMsg16[43].Q;			OUT_CU.bMsg1643 :=	xMsg16[43].Q;
	MM2VIS.bMsg1644 :=	xMsg16[44].Q;			OUT_CU.bMsg1644 :=	xMsg16[44].Q;
	MM2VIS.bMsg1645 :=	xMsg16[45].Q;			OUT_CU.bMsg1645 :=	xMsg16[45].Q;
	MM2VIS.bMsg1646 :=	xMsg16[46].Q;			OUT_CU.bMsg1646 :=	xMsg16[46].Q;
	MM2VIS.bMsg1647 :=	xMsg16[47].Q;			OUT_CU.bMsg1647 :=	xMsg16[47].Q;
	MM2VIS.bMsg1648 :=	xMsg16[48].Q;			OUT_CU.bMsg1648 :=	xMsg16[48].Q;
	MM2VIS.bMsg1649 :=	xMsg16[49].Q;			OUT_CU.bMsg1649 :=	xMsg16[49].Q;
	MM2VIS.bMsg1650 :=	xMsg16[50].Q;			OUT_CU.bMsg1650 :=	xMsg16[50].Q;

	MM2VIS.bMsg1651 :=	xMsg16[51].Q;			OUT_CU.bMsg1651 :=	xMsg16[51].Q;
	MM2VIS.bMsg1652 :=	xMsg16[52].Q;			OUT_CU.bMsg1652 :=	xMsg16[52].Q;
	MM2VIS.bMsg1653 :=	xMsg16[53].Q;			OUT_CU.bMsg1653 :=	xMsg16[53].Q;
	MM2VIS.bMsg1654 :=	xMsg16[54].Q;			OUT_CU.bMsg1654 :=	xMsg16[54].Q;
	MM2VIS.bMsg1655 :=	xMsg16[55].Q;			OUT_CU.bMsg1655 :=	xMsg16[55].Q;
	MM2VIS.bMsg1656 :=	xMsg16[56].Q;			OUT_CU.bMsg1656 :=	xMsg16[56].Q;
	MM2VIS.bMsg1657 :=	xMsg16[57].Q;			OUT_CU.bMsg1657 :=	xMsg16[57].Q;
	MM2VIS.bMsg1658 :=	xMsg16[58].Q;			OUT_CU.bMsg1658 :=	xMsg16[58].Q;
	MM2VIS.bMsg1659 :=	xMsg16[59].Q;			OUT_CU.bMsg1659 :=	xMsg16[59].Q;
	MM2VIS.bMsg1660 :=	xMsg16[60].Q;			OUT_CU.bMsg1660 :=	xMsg16[60].Q;

	MM2VIS.bMsg1661 :=	xMsg16[61].Q;			OUT_CU.bMsg1661 :=	xMsg16[61].Q;
	MM2VIS.bMsg1662 :=	xMsg16[62].Q;			OUT_CU.bMsg1662 :=	xMsg16[62].Q;
	MM2VIS.bMsg1663 :=	xMsg16[63].Q;			OUT_CU.bMsg1663 :=	xMsg16[63].Q;
	MM2VIS.bMsg1664 :=	xMsg16[64].Q;			OUT_CU.bMsg1664 :=	xMsg16[64].Q;
	MM2VIS.bMsg1665 :=	xMsg16[65].Q;			OUT_CU.bMsg1665 :=	xMsg16[65].Q;
	MM2VIS.bMsg1666 :=	xMsg16[66].Q;			OUT_CU.bMsg1666 :=	xMsg16[66].Q;
	MM2VIS.bMsg1667 :=	xMsg16[67].Q;			OUT_CU.bMsg1667 :=	xMsg16[67].Q;
	MM2VIS.bMsg1668 :=	xMsg16[68].Q;			OUT_CU.bMsg1668 :=	xMsg16[68].Q;
	MM2VIS.bMsg1669 :=	xMsg16[69].Q;			OUT_CU.bMsg1669 :=	xMsg16[69].Q;
	MM2VIS.bMsg1670 :=	xMsg16[70].Q;			OUT_CU.bMsg1670 :=	xMsg16[70].Q;

	MM2VIS.bMsg1671 :=	xMsg16[71].Q;			OUT_CU.bMsg1671 :=	xMsg16[71].Q;
	MM2VIS.bMsg1672 :=	xMsg16[72].Q;			OUT_CU.bMsg1672 :=	xMsg16[72].Q;
	MM2VIS.bMsg1673 :=	xMsg16[73].Q;			OUT_CU.bMsg1673 :=	xMsg16[73].Q;
	MM2VIS.bMsg1674 :=	xMsg16[74].Q;			OUT_CU.bMsg1674 :=	xMsg16[74].Q;
	MM2VIS.bMsg1675 :=	xMsg16[75].Q;			OUT_CU.bMsg1675 :=	xMsg16[75].Q;
	MM2VIS.bMsg1676 :=	xMsg16[76].Q;			OUT_CU.bMsg1676 :=	xMsg16[76].Q;
	MM2VIS.bMsg1677 :=	xMsg16[77].Q;			OUT_CU.bMsg1677 :=	xMsg16[77].Q;
	MM2VIS.bMsg1678 :=	xMsg16[78].Q;			OUT_CU.bMsg1678 :=	xMsg16[78].Q;
	MM2VIS.bMsg1679 :=	xMsg16[79].Q;			OUT_CU.bMsg1679 :=	xMsg16[79].Q;
	MM2VIS.bMsg1680 :=	xMsg16[80].Q;			OUT_CU.bMsg1680 :=	xMsg16[80].Q;

	MM2VIS.bMsg1681 :=	xMsg16[81].Q;			OUT_CU.bMsg1681 :=	xMsg16[81].Q;
	MM2VIS.bMsg1682 :=	xMsg16[82].Q;			OUT_CU.bMsg1682 :=	xMsg16[82].Q;
	MM2VIS.bMsg1683 :=	xMsg16[83].Q;			OUT_CU.bMsg1683 :=	xMsg16[83].Q;
	MM2VIS.bMsg1684 :=	xMsg16[84].Q;			OUT_CU.bMsg1684 :=	xMsg16[84].Q;
	MM2VIS.bMsg1685 :=	xMsg16[85].Q;			OUT_CU.bMsg1685 :=	xMsg16[85].Q;
	MM2VIS.bMsg1686 :=	xMsg16[86].Q;			OUT_CU.bMsg1686 :=	xMsg16[86].Q;
	MM2VIS.bMsg1687 :=	xMsg16[87].Q;			OUT_CU.bMsg1687 :=	xMsg16[87].Q;
	MM2VIS.bMsg1688 :=	xMsg16[88].Q;			OUT_CU.bMsg1688 :=	xMsg16[88].Q;
	MM2VIS.bMsg1689 :=	xMsg16[89].Q;			OUT_CU.bMsg1689 :=	xMsg16[89].Q;
	MM2VIS.bMsg1690 :=	xMsg16[90].Q;			OUT_CU.bMsg1690 :=	xMsg16[90].Q;

	MM2VIS.bMsg1691 :=	xMsg16[91].Q;			OUT_CU.bMsg1691 :=	xMsg16[91].Q;
	MM2VIS.bMsg1692 :=	xMsg16[92].Q;			OUT_CU.bMsg1692 :=	xMsg16[92].Q;
	MM2VIS.bMsg1693 :=	xMsg16[93].Q;			OUT_CU.bMsg1693 :=	xMsg16[93].Q;
	MM2VIS.bMsg1694 :=	xMsg16[94].Q;			OUT_CU.bMsg1694 :=	xMsg16[94].Q;
	MM2VIS.bMsg1695 :=	xMsg16[95].Q;			OUT_CU.bMsg1695 :=	xMsg16[95].Q;
	MM2VIS.bMsg1696 :=	xMsg16[96].Q;			OUT_CU.bMsg1696 :=	xMsg16[96].Q;
	MM2VIS.bMsg1697 :=	xMsg16[97].Q;			OUT_CU.bMsg1697 :=	xMsg16[97].Q;
	MM2VIS.bMsg1698 :=	xMsg16[98].Q;			OUT_CU.bMsg1698 :=	xMsg16[98].Q;
												OUT_CU.bMsg1699 :=	xMsg16[99].Q; 	(*remove duplicate MM2VIS handling*)
												OUT_CU.bMsg1700 :=	xMsg16[100].Q;  (*remove duplicate MM2VIS handling*)

	(* Forwarding of spare warning messages: *)
	MM2VIS.bMsg1701 :=	xMsg17[01].Q;			OUT_CU.bMsg1701 :=	xMsg17[01].Q;  	(*do not remove 1701-*)
	MM2VIS.bMsg1702 :=	xMsg17[02].Q;			OUT_CU.bMsg1702 :=	xMsg17[02].Q;
	MM2VIS.bMsg1703 :=	xMsg17[03].Q;			OUT_CU.bMsg1703 :=	xMsg17[03].Q;
	MM2VIS.bMsg1704 :=	xMsg17[04].Q;			OUT_CU.bMsg1704 :=	xMsg17[04].Q;
	MM2VIS.bMsg1705 :=	xMsg17[05].Q;			OUT_CU.bMsg1705 :=	xMsg17[05].Q;
	MM2VIS.bMsg1706 :=	xMsg17[06].Q;			OUT_CU.bMsg1706 :=	xMsg17[06].Q;
	MM2VIS.bMsg1707 :=	xMsg17[07].Q;			OUT_CU.bMsg1707 :=	xMsg17[07].Q;
	MM2VIS.bMsg1708 :=	xMsg17[08].Q;			OUT_CU.bMsg1708 :=	xMsg17[08].Q;
	MM2VIS.bMsg1709 :=	xMsg17[09].Q;			OUT_CU.bMsg1709 :=	xMsg17[09].Q;
	MM2VIS.bMsg1710 :=	xMsg17[10].Q;			OUT_CU.bMsg1710 :=	xMsg17[10].Q;

	MM2VIS.bMsg1711 :=	xMsg17[11].Q;			OUT_CU.bMsg1711 :=	xMsg17[11].Q;
	MM2VIS.bMsg1712 :=	xMsg17[12].Q;			OUT_CU.bMsg1712 :=	xMsg17[12].Q;
	MM2VIS.bMsg1713 :=	xMsg17[13].Q;			OUT_CU.bMsg1713 :=	xMsg17[13].Q;
	MM2VIS.bMsg1714 :=	xMsg17[14].Q;			OUT_CU.bMsg1714 :=	xMsg17[14].Q;
	MM2VIS.bMsg1715 :=	xMsg17[15].Q;			OUT_CU.bMsg1715 :=	xMsg17[15].Q;
	MM2VIS.bMsg1716 :=	xMsg17[16].Q;			OUT_CU.bMsg1716 :=	xMsg17[16].Q;
	MM2VIS.bMsg1717 :=	xMsg17[17].Q;			OUT_CU.bMsg1717 :=	xMsg17[17].Q;
	MM2VIS.bMsg1718 :=	xMsg17[18].Q;			OUT_CU.bMsg1718 :=	xMsg17[18].Q;
	MM2VIS.bMsg1719 :=	xMsg17[19].Q;			OUT_CU.bMsg1719 :=	xMsg17[19].Q;
	MM2VIS.bMsg1720 :=	xMsg17[20].Q;			OUT_CU.bMsg1720 :=	xMsg17[20].Q;

	MM2VIS.bMsg1721 :=	xMsg17[21].Q;			OUT_CU.bMsg1721 :=	xMsg17[21].Q;
	MM2VIS.bMsg1722 :=	xMsg17[22].Q;			OUT_CU.bMsg1722 :=	xMsg17[22].Q;
	MM2VIS.bMsg1723 :=	xMsg17[23].Q;			OUT_CU.bMsg1723 :=	xMsg17[23].Q;
	MM2VIS.bMsg1724 :=	xMsg17[24].Q;			OUT_CU.bMsg1724 :=	xMsg17[24].Q;
	MM2VIS.bMsg1725 :=	xMsg17[25].Q;			OUT_CU.bMsg1725 :=	xMsg17[25].Q;
	MM2VIS.bMsg1726 :=	xMsg17[26].Q;			OUT_CU.bMsg1726 :=	xMsg17[26].Q;
	MM2VIS.bMsg1727 :=	xMsg17[27].Q;			OUT_CU.bMsg1727 :=	xMsg17[27].Q;
	MM2VIS.bMsg1728 :=	xMsg17[28].Q;			OUT_CU.bMsg1728 :=	xMsg17[28].Q;
	MM2VIS.bMsg1729 :=	xMsg17[29].Q;			OUT_CU.bMsg1729 :=	xMsg17[29].Q;
	MM2VIS.bMsg1730 :=	xMsg17[30].Q;			OUT_CU.bMsg1730 :=	xMsg17[30].Q;

	MM2VIS.bMsg1731 :=	xMsg17[31].Q;			OUT_CU.bMsg1731 :=	xMsg17[31].Q;
	MM2VIS.bMsg1732 :=	xMsg17[32].Q;			OUT_CU.bMsg1732 :=	xMsg17[32].Q;
	MM2VIS.bMsg1733 :=	xMsg17[33].Q;			OUT_CU.bMsg1733 :=	xMsg17[33].Q;
	MM2VIS.bMsg1734 :=	xMsg17[34].Q;			OUT_CU.bMsg1734 :=	xMsg17[34].Q;
	MM2VIS.bMsg1735 :=	xMsg17[35].Q;			OUT_CU.bMsg1735 :=	xMsg17[35].Q;
	MM2VIS.bMsg1736 :=	xMsg17[36].Q;			OUT_CU.bMsg1736 :=	xMsg17[36].Q;
	MM2VIS.bMsg1737 :=	xMsg17[37].Q;			OUT_CU.bMsg1737 :=	xMsg17[37].Q;
	MM2VIS.bMsg1738 :=	xMsg17[38].Q;			OUT_CU.bMsg1738 :=	xMsg17[38].Q;
	MM2VIS.bMsg1739 :=	xMsg17[39].Q;			OUT_CU.bMsg1739 :=	xMsg17[39].Q;
	MM2VIS.bMsg1740 :=	xMsg17[40].Q;			OUT_CU.bMsg1740 :=	xMsg17[40].Q;

	MM2VIS.bMsg1741 :=	xMsg17[41].Q;			OUT_CU.bMsg1741 :=	xMsg17[41].Q;
	MM2VIS.bMsg1742 :=	xMsg17[42].Q;			OUT_CU.bMsg1742 :=	xMsg17[42].Q;
	MM2VIS.bMsg1743 :=	xMsg17[43].Q;			OUT_CU.bMsg1743 :=	xMsg17[43].Q;
	MM2VIS.bMsg1744 :=	xMsg17[44].Q;			OUT_CU.bMsg1744 :=	xMsg17[44].Q;
	MM2VIS.bMsg1745 :=	xMsg17[45].Q;			OUT_CU.bMsg1745 :=	xMsg17[45].Q;
	MM2VIS.bMsg1746 :=	xMsg17[46].Q;			OUT_CU.bMsg1746 :=	xMsg17[46].Q;
	MM2VIS.bMsg1747 :=	xMsg17[47].Q;			OUT_CU.bMsg1747 :=	xMsg17[47].Q;
	MM2VIS.bMsg1748 :=	xMsg17[48].Q;			OUT_CU.bMsg1748 :=	xMsg17[48].Q;
	MM2VIS.bMsg1749 :=	xMsg17[49].Q;			OUT_CU.bMsg1749 :=	xMsg17[49].Q;
	MM2VIS.bMsg1750 :=	xMsg17[50].Q;			OUT_CU.bMsg1750 :=	xMsg17[50].Q;

	MM2VIS.bMsg1751 :=	xMsg17[51].Q;			OUT_CU.bMsg1751 :=	xMsg17[51].Q;
	MM2VIS.bMsg1752 :=	xMsg17[52].Q;			OUT_CU.bMsg1752 :=	xMsg17[52].Q;
	MM2VIS.bMsg1753 :=	xMsg17[53].Q;			OUT_CU.bMsg1753 :=	xMsg17[53].Q;
	MM2VIS.bMsg1754 :=	xMsg17[54].Q;			OUT_CU.bMsg1754 :=	xMsg17[54].Q;
	MM2VIS.bMsg1755 :=	xMsg17[55].Q;			OUT_CU.bMsg1755 :=	xMsg17[55].Q;
	MM2VIS.bMsg1756 :=	xMsg17[56].Q;			OUT_CU.bMsg1756 :=	xMsg17[56].Q;
	MM2VIS.bMsg1757 :=	xMsg17[57].Q;			OUT_CU.bMsg1757 :=	xMsg17[57].Q;
	MM2VIS.bMsg1758 :=	xMsg17[58].Q;			OUT_CU.bMsg1758 :=	xMsg17[58].Q;
	MM2VIS.bMsg1759 :=	xMsg17[59].Q;			OUT_CU.bMsg1759 :=	xMsg17[59].Q;
	MM2VIS.bMsg1760 :=	xMsg17[60].Q;			OUT_CU.bMsg1760 :=	xMsg17[60].Q;

	MM2VIS.bMsg1761 :=	xMsg17[61].Q;			OUT_CU.bMsg1761 :=	xMsg17[61].Q;
	MM2VIS.bMsg1762 :=	xMsg17[62].Q;			OUT_CU.bMsg1762 :=	xMsg17[62].Q;
	MM2VIS.bMsg1763 :=	xMsg17[63].Q;			OUT_CU.bMsg1763 :=	xMsg17[63].Q;
	MM2VIS.bMsg1764 :=	xMsg17[64].Q;			OUT_CU.bMsg1764 :=	xMsg17[64].Q;
	MM2VIS.bMsg1765 :=	xMsg17[65].Q;			OUT_CU.bMsg1765 :=	xMsg17[65].Q;
	MM2VIS.bMsg1766 :=	xMsg17[66].Q;			OUT_CU.bMsg1766 :=	xMsg17[66].Q;
	MM2VIS.bMsg1767 :=	xMsg17[67].Q;			OUT_CU.bMsg1767 :=	xMsg17[67].Q;
	MM2VIS.bMsg1768 :=	xMsg17[68].Q;			OUT_CU.bMsg1768 :=	xMsg17[68].Q;
	MM2VIS.bMsg1769 :=	xMsg17[69].Q;			OUT_CU.bMsg1769 :=	xMsg17[69].Q;
	MM2VIS.bMsg1770 :=	xMsg17[70].Q;			OUT_CU.bMsg1770 :=	xMsg17[70].Q;

	MM2VIS.bMsg1771 :=	xMsg17[71].Q;			OUT_CU.bMsg1771 :=	xMsg17[71].Q;
	MM2VIS.bMsg1772 :=	xMsg17[72].Q;			OUT_CU.bMsg1772 :=	xMsg17[72].Q;
	MM2VIS.bMsg1773 :=	xMsg17[73].Q;			OUT_CU.bMsg1773 :=	xMsg17[73].Q;
	MM2VIS.bMsg1774 :=	xMsg17[74].Q;			OUT_CU.bMsg1774 :=	xMsg17[74].Q;
	MM2VIS.bMsg1775 :=	xMsg17[75].Q;			OUT_CU.bMsg1775 :=	xMsg17[75].Q;
	MM2VIS.bMsg1776 :=	xMsg17[76].Q;			OUT_CU.bMsg1776 :=	xMsg17[76].Q;
	MM2VIS.bMsg1777 :=	xMsg17[77].Q;			OUT_CU.bMsg1777 :=	xMsg17[77].Q;
	MM2VIS.bMsg1778 :=	xMsg17[78].Q;			OUT_CU.bMsg1778 :=	xMsg17[78].Q;
	MM2VIS.bMsg1779 :=	xMsg17[79].Q;			OUT_CU.bMsg1779 :=	xMsg17[79].Q;
	MM2VIS.bMsg1780 :=	xMsg17[80].Q;			OUT_CU.bMsg1780 :=	xMsg17[80].Q;

	MM2VIS.bMsg1781 :=	xMsg17[81].Q;			OUT_CU.bMsg1781 :=	xMsg17[81].Q;
	MM2VIS.bMsg1782 :=	xMsg17[82].Q;			OUT_CU.bMsg1782 :=	xMsg17[82].Q;
	MM2VIS.bMsg1783 :=	xMsg17[83].Q;			OUT_CU.bMsg1783 :=	xMsg17[83].Q;
	MM2VIS.bMsg1784 :=	xMsg17[84].Q;			OUT_CU.bMsg1784 :=	xMsg17[84].Q;
	MM2VIS.bMsg1785 :=	xMsg17[85].Q;			OUT_CU.bMsg1785 :=	xMsg17[85].Q;
	MM2VIS.bMsg1786 :=	xMsg17[86].Q;			OUT_CU.bMsg1786 :=	xMsg17[86].Q;
	MM2VIS.bMsg1787 :=	xMsg17[87].Q;			OUT_CU.bMsg1787 :=	xMsg17[87].Q;
	MM2VIS.bMsg1788 :=	xMsg17[88].Q;			OUT_CU.bMsg1788 :=	xMsg17[88].Q;
	MM2VIS.bMsg1789 :=	xMsg17[89].Q;			OUT_CU.bMsg1789 :=	xMsg17[89].Q;
	MM2VIS.bMsg1790 :=	xMsg17[90].Q;			OUT_CU.bMsg1790 :=	xMsg17[90].Q;

	MM2VIS.bMsg1791 :=	xMsg17[91].Q;			OUT_CU.bMsg1791 :=	xMsg17[91].Q;
	MM2VIS.bMsg1792 :=	xMsg17[92].Q;			OUT_CU.bMsg1792 :=	xMsg17[92].Q;
	MM2VIS.bMsg1793 :=	xMsg17[93].Q;			OUT_CU.bMsg1793 :=	xMsg17[93].Q;
	MM2VIS.bMsg1794 :=	xMsg17[94].Q;			OUT_CU.bMsg1794 :=	xMsg17[94].Q;
	MM2VIS.bMsg1795 :=	xMsg17[95].Q;			OUT_CU.bMsg1795 :=	xMsg17[95].Q;
	MM2VIS.bMsg1796 :=	xMsg17[96].Q;			OUT_CU.bMsg1796 :=	xMsg17[96].Q;
	MM2VIS.bMsg1797 :=	xMsg17[97].Q;			OUT_CU.bMsg1797 :=	xMsg17[97].Q;
	MM2VIS.bMsg1798 :=	xMsg17[98].Q;			OUT_CU.bMsg1798 :=	xMsg17[98].Q;
	MM2VIS.bMsg1799 :=	xMsg17[99].Q;			OUT_CU.bMsg1799 :=	xMsg17[99].Q;
	MM2VIS.bMsg1800 :=	xMsg17[100].Q;			OUT_CU.bMsg1800 :=	xMsg17[100].Q;		(*!corr.!*)

	MM2VIS.bMsg8701 :=	OUT_CU.bMsg8701 :=	xMsg87[01].Q;	 (*import HMI Extension *)
	MM2VIS.bMsg8702 :=	OUT_CU.bMsg8702 :=	xMsg87[02].Q;	 (*import HMI Extension *)
	MM2VIS.bMsg8703 :=	OUT_CU.bMsg8703 :=	xMsg87[03].Q;	 (*import HMI Extension *)
	MM2VIS.bMsg8704 :=	OUT_CU.bMsg8704 :=	xMsg87[04].Q;	 (*import HMI Extension *)
	MM2VIS.bMsg8705 :=	OUT_CU.bMsg8705 :=	xMsg87[05].Q;	 (*import HMI Extension *)
	MM2VIS.bMsg8706 :=	OUT_CU.bMsg8706 :=	xMsg87[06].Q;	 (*import HMI Extension *)
	MM2VIS.bMsg8707 :=	OUT_CU.bMsg8707 :=	xMsg87[07].Q;	 (*import HMI Extension *)
	MM2VIS.bMsg8708 :=	OUT_CU.bMsg8708 :=	xMsg87[08].Q;	 (*import HMI Extension *)
	MM2VIS.bMsg8709 :=	OUT_CU.bMsg8709 :=	xMsg87[09].Q;	 (*import HMI Extension *)
	MM2VIS.bMsg8710 :=	OUT_CU.bMsg8710 :=	xMsg87[10].Q;	 (*import HMI Extension *)

	MM2VIS.bMsg8711 :=	OUT_CU.bMsg8711 :=	xMsg87[11].Q;	 (*import HMI Extension *)
	MM2VIS.bMsg8712 :=	OUT_CU.bMsg8712 :=	xMsg87[12].Q;	 (*import HMI Extension *)
	MM2VIS.bMsg8713 :=	OUT_CU.bMsg8713 :=	xMsg87[13].Q;	 (*import HMI Extension *)
	MM2VIS.bMsg8714 :=	OUT_CU.bMsg8714 :=	xMsg87[14].Q;	 (*import HMI Extension *)
	MM2VIS.bMsg8715 :=	OUT_CU.bMsg8715 :=	xMsg87[15].Q;	 (*import HMI Extension *)
	MM2VIS.bMsg8716 :=	OUT_CU.bMsg8716 :=	xMsg87[16].Q;	 (*import HMI Extension *)
	MM2VIS.bMsg8717 :=	OUT_CU.bMsg8717 :=	xMsg87[17].Q;	 (*import HMI Extension *)
	MM2VIS.bMsg8718 :=	OUT_CU.bMsg8718 :=	xMsg87[18].Q;	 (*import HMI Extension *)
	MM2VIS.bMsg8719 :=	OUT_CU.bMsg8719 :=	xMsg87[19].Q;	 (*import HMI Extension *)
	MM2VIS.bMsg8720 :=	OUT_CU.bMsg8720 :=	xMsg87[20].Q;	 (*import HMI Extension *)

	MM2VIS.bMsg8721 :=	OUT_CU.bMsg8721 :=	xMsg87[21].Q;	 (*import HMI Extension *)
	MM2VIS.bMsg8722 :=	OUT_CU.bMsg8722 :=	xMsg87[22].Q;	 (*import HMI Extension *)
	MM2VIS.bMsg8723 :=	OUT_CU.bMsg8723 :=	xMsg87[23].Q;	 (*import HMI Extension *)
	MM2VIS.bMsg8724 :=	OUT_CU.bMsg8724 :=	xMsg87[24].Q;	 (*import HMI Extension *)
	MM2VIS.bMsg8725 :=	OUT_CU.bMsg8725 :=	xMsg87[25].Q;	 (*import HMI Extension *)
	MM2VIS.bMsg8726 :=	OUT_CU.bMsg8726 :=	xMsg87[26].Q;	 (*import HMI Extension *)
	MM2VIS.bMsg8727 :=	OUT_CU.bMsg8727 :=	xMsg87[27].Q;	 (*import HMI Extension *)
	MM2VIS.bMsg8728 :=	OUT_CU.bMsg8728 :=	xMsg87[28].Q;	 (*import HMI Extension *)
	MM2VIS.bMsg8729 :=	OUT_CU.bMsg8729 :=	xMsg87[29].Q;	 (*import HMI Extension *)
	MM2VIS.bMsg8730 :=	OUT_CU.bMsg8730 :=	xMsg87[30].Q;	 (*import HMI Extension *)

	MM2VIS.bMsg8731 :=	OUT_CU.bMsg8731 :=	xMsg87[31].Q;	 (*import HMI Extension *)
	MM2VIS.bMsg8732 :=	OUT_CU.bMsg8732 :=	xMsg87[32].Q;	 (*import HMI Extension *)
	MM2VIS.bMsg8733 :=	OUT_CU.bMsg8733 :=	xMsg87[33].Q;	 (*import HMI Extension *)
	MM2VIS.bMsg8734 :=	OUT_CU.bMsg8734 :=	xMsg87[34].Q;	 (*import HMI Extension *)
	MM2VIS.bMsg8735 :=	OUT_CU.bMsg8735 :=	xMsg87[35].Q;	 (*import HMI Extension *)
	MM2VIS.bMsg8736 :=	OUT_CU.bMsg8736 :=	xMsg87[36].Q;	 (*import HMI Extension *)
	MM2VIS.bMsg8737 :=	OUT_CU.bMsg8737 :=	xMsg87[37].Q;	 (*import HMI Extension *)
	MM2VIS.bMsg8738 :=	OUT_CU.bMsg8738 :=	xMsg87[38].Q;	 (*import HMI Extension *)
	MM2VIS.bMsg8739 :=	OUT_CU.bMsg8739 :=	xMsg87[39].Q;	 (*import HMI Extension *)
	MM2VIS.bMsg8740 :=	OUT_CU.bMsg8740 :=	xMsg87[40].Q;	 (*import HMI Extension *)

	MM2VIS.bMsg8741 :=	OUT_CU.bMsg8741 :=	xMsg87[41].Q;	 (*import HMI Extension *)
	MM2VIS.bMsg8742 :=	OUT_CU.bMsg8742 :=	xMsg87[42].Q;	 (*import HMI Extension *)
	MM2VIS.bMsg8743 :=	OUT_CU.bMsg8743 :=	xMsg87[43].Q;	 (*import HMI Extension *)
	MM2VIS.bMsg8744 :=	OUT_CU.bMsg8744 :=	xMsg87[44].Q;	 (*import HMI Extension *)
	MM2VIS.bMsg8745 :=	OUT_CU.bMsg8745 :=	xMsg87[45].Q;	 (*import HMI Extension *)
	MM2VIS.bMsg8746 :=	OUT_CU.bMsg8746 :=	xMsg87[46].Q;	 (*import HMI Extension *)
	MM2VIS.bMsg8747 :=	OUT_CU.bMsg8747 :=	xMsg87[47].Q;	 (*import HMI Extension *)
	MM2VIS.bMsg8748 :=	OUT_CU.bMsg8748 :=	xMsg87[48].Q;	 (*import HMI Extension *)
	MM2VIS.bMsg8749 :=	OUT_CU.bMsg8749 :=	xMsg87[49].Q;	 (*import HMI Extension *)
	MM2VIS.bMsg8750 :=	OUT_CU.bMsg8750 :=	xMsg87[50].Q;	 (*import HMI Extension *)

	MM2VIS.bMsg8751 :=	OUT_CU.bMsg8751 :=	xMsg87[51].Q;	 (*import HMI Extension *)
	MM2VIS.bMsg8752 :=	OUT_CU.bMsg8752 :=	xMsg87[52].Q;	 (*import HMI Extension *)
	MM2VIS.bMsg8753 :=	OUT_CU.bMsg8753 :=	xMsg87[53].Q;	 (*import HMI Extension *)
	MM2VIS.bMsg8754 :=	OUT_CU.bMsg8754 :=	xMsg87[54].Q;	 (*import HMI Extension *)
	MM2VIS.bMsg8755 :=	OUT_CU.bMsg8755 :=	xMsg87[55].Q;	 (*import HMI Extension *)
	MM2VIS.bMsg8756 :=	OUT_CU.bMsg8756 :=	xMsg87[56].Q;	 (*import HMI Extension *)
	MM2VIS.bMsg8757 :=	OUT_CU.bMsg8757 :=	xMsg87[57].Q;	 (*import HMI Extension *)
	MM2VIS.bMsg8758 :=	OUT_CU.bMsg8758 :=	xMsg87[58].Q;	 (*import HMI Extension *)
	MM2VIS.bMsg8759 :=	OUT_CU.bMsg8759 :=	xMsg87[59].Q;	 (*import HMI Extension *)
	MM2VIS.bMsg8760 :=	OUT_CU.bMsg8760 :=	xMsg87[60].Q;	 (*import HMI Extension *)

	MM2VIS.bMsg8761 :=	OUT_CU.bMsg8761 :=	xMsg87[61].Q;	 (*import HMI Extension *)
	MM2VIS.bMsg8762 :=	OUT_CU.bMsg8762 :=	xMsg87[62].Q;	 (*import HMI Extension *)
	MM2VIS.bMsg8763 :=	OUT_CU.bMsg8763 :=	xMsg87[63].Q;	 (*import HMI Extension *)
	MM2VIS.bMsg8764 :=	OUT_CU.bMsg8764 :=	xMsg87[64].Q;	 (*import HMI Extension *)
	MM2VIS.bMsg8765 :=	OUT_CU.bMsg8765 :=	xMsg87[65].Q;	 (*import HMI Extension *)
	MM2VIS.bMsg8766 :=	OUT_CU.bMsg8766 :=	xMsg87[66].Q;	 (*import HMI Extension *)
	MM2VIS.bMsg8767 :=	OUT_CU.bMsg8767 :=	xMsg87[67].Q;	 (*import HMI Extension *)
	MM2VIS.bMsg8768 :=	OUT_CU.bMsg8768 :=	xMsg87[68].Q;	 (*import HMI Extension *)
	MM2VIS.bMsg8769 :=	OUT_CU.bMsg8769 :=	xMsg87[69].Q;	 (*import HMI Extension *)
	MM2VIS.bMsg8770 :=	OUT_CU.bMsg8770 :=	xMsg87[70].Q;	 (*import HMI Extension *)

	MM2VIS.bMsg8771 :=	OUT_CU.bMsg8771 :=	xMsg87[71].Q;	 (*import HMI Extension *)
	MM2VIS.bMsg8772 :=	OUT_CU.bMsg8772 :=	xMsg87[72].Q;	 (*import HMI Extension *)
	MM2VIS.bMsg8773 :=	OUT_CU.bMsg8773 :=	xMsg87[73].Q;	 (*import HMI Extension *)
	MM2VIS.bMsg8774 :=	OUT_CU.bMsg8774 :=	xMsg87[74].Q;	 (*import HMI Extension *)
	MM2VIS.bMsg8775 :=	OUT_CU.bMsg8775 :=	xMsg87[75].Q;	 (*import HMI Extension *)
	MM2VIS.bMsg8776 :=	OUT_CU.bMsg8776 :=	xMsg87[76].Q;	 (*import HMI Extension *)
	MM2VIS.bMsg8777 :=	OUT_CU.bMsg8777 :=	xMsg87[77].Q;	 (*import HMI Extension *)
	MM2VIS.bMsg8778 :=	OUT_CU.bMsg8778 :=	xMsg87[78].Q;	 (*import HMI Extension *)
	MM2VIS.bMsg8779 :=	OUT_CU.bMsg8779 :=	xMsg87[79].Q;	 (*import HMI Extension *)
	MM2VIS.bMsg8780 :=	OUT_CU.bMsg8780 :=	xMsg87[80].Q;	 (*import HMI Extension *)

	MM2VIS.bMsg8781 :=	OUT_CU.bMsg8781 :=	xMsg87[81].Q;	 (*import HMI Extension *)
	MM2VIS.bMsg8782 :=	OUT_CU.bMsg8782 :=	xMsg87[82].Q;	 (*import HMI Extension *)
	MM2VIS.bMsg8783 :=	OUT_CU.bMsg8783 :=	xMsg87[83].Q;	 (*import HMI Extension *)
	MM2VIS.bMsg8784 :=	OUT_CU.bMsg8784 :=	xMsg87[84].Q;	 (*import HMI Extension *)
	MM2VIS.bMsg8785 :=	OUT_CU.bMsg8785 :=	xMsg87[85].Q;	 (*import HMI Extension *)
	MM2VIS.bMsg8786 :=	OUT_CU.bMsg8786 :=	xMsg87[86].Q;	 (*import HMI Extension *)
	MM2VIS.bMsg8787 :=	OUT_CU.bMsg8787 :=	xMsg87[87].Q;	 (*import HMI Extension *)
	MM2VIS.bMsg8788 :=	OUT_CU.bMsg8788 :=	xMsg87[88].Q;	 (*import HMI Extension *)
	MM2VIS.bMsg8789 :=	OUT_CU.bMsg8789 :=	xMsg87[89].Q;	 (*import HMI Extension *)
	MM2VIS.bMsg8790 :=	OUT_CU.bMsg8790 :=	xMsg87[90].Q;	 (*import HMI Extension *)

	MM2VIS.bMsg8791 :=	OUT_CU.bMsg8791 :=	xMsg87[91].Q;	 (*import HMI Extension *)
	MM2VIS.bMsg8792 :=	OUT_CU.bMsg8792 :=	xMsg87[92].Q;	 (*import HMI Extension *)
	MM2VIS.bMsg8793 :=	OUT_CU.bMsg8793 :=	xMsg87[93].Q;	 (*import HMI Extension *)
	MM2VIS.bMsg8794 :=	OUT_CU.bMsg8794 :=	xMsg87[94].Q;	 (*import HMI Extension *)
	MM2VIS.bMsg8795 :=	OUT_CU.bMsg8795 :=	xMsg87[95].Q;	 (*import HMI Extension *)
	MM2VIS.bMsg8796 :=	OUT_CU.bMsg8796 :=	xMsg87[96].Q;	 (*import HMI Extension *)
	MM2VIS.bMsg8797 :=	OUT_CU.bMsg8797 :=	xMsg87[97].Q;	 (*import HMI Extension *)
	MM2VIS.bMsg8798 :=	OUT_CU.bMsg8798 :=	xMsg87[98].Q;	 (*import HMI Extension *)
	MM2VIS.bMsg8799 :=	OUT_CU.bMsg8799 :=	xMsg87[99].Q;	 (*import HMI Extension *)
(*	MM2VIS.bMsg4300 :=	OUT_CU.bMsg4300 :=	xMsg87[100].Q;	 (*import HMI Extension  OLD do not use anymore *)

	(* forwarding of operating messages  *)

	xMsg3232.Enable		:=	IN_CU.tPB2MM.bParaSetupOk ;
	xMsg3232.Set		:=	OUT_CU.bMsg3232;		(* B3232 reserve operating message 1 *)
	IF xMsg3232.Set THEN iReset_Msg3232 := iDelay_MsgAutoReset_100ms; ELSE iReset_Msg3232 := LIMIT(0, iReset_Msg3232 -1,32767); END_IF		(* activate 'Message Hold Time' to avoid log clathering by repeated OpMsg entries *)
	xMsg3232.Reset 		:= 	iReset_Msg3232 < 1;		//.Reset := TRUE;
	xMsg3232();
	MM2VIS.bMsg3232		:=	xMsg3232.Q;

	xMsg3233.Enable		:=	IN_CU.tPB2MM.bParaSetupOk ;
	xMsg3233.Set		:=	OUT_CU.bMsg3233;		(* B3233 reserve operating message 2 *)
	IF xMsg3233.Set THEN iReset_Msg3233 := iDelay_MsgAutoReset_100ms; ELSE iReset_Msg3233 := LIMIT(0, iReset_Msg3233 -1,32767); END_IF		(* activate 'Message Hold Time' to avoid log clathering by repeated OpMsg entries *)
	xMsg3233.Reset 		:= 	iReset_Msg3233 < 1;		//.Reset := TRUE;
	xMsg3233();
	MM2VIS.bMsg3233		:=	xMsg3233.Q;

	xMsg3234.Enable		:=	IN_CU.tPB2MM.bParaSetupOk ;
	xMsg3234.Set		:=	OUT_CU.bMsg3234;		(* B3234 reserve operating message 3 *)
	IF xMsg3234.Set THEN iReset_Msg3234 := iDelay_MsgAutoReset_100ms; ELSE iReset_Msg3234 := LIMIT(0, iReset_Msg3234 -1,32767); END_IF		(* activate 'Message Hold Time' to avoid log clathering by repeated OpMsg entries *)
	xMsg3234.Reset 		:= 	iReset_Msg3234 < 1;		//.Reset := TRUE;
	xMsg3234();
	MM2VIS.bMsg3234		:=	xMsg3234.Q;

	xMsg3235.Enable		:=	IN_CU.tPB2MM.bParaSetupOk ;
	xMsg3235.Set		:=	OUT_CU.bMsg3235;		(* B3235 reserve operating message 4 *)
	IF xMsg3235.Set THEN iReset_Msg3235 := iDelay_MsgAutoReset_100ms; ELSE iReset_Msg3235 := LIMIT(0, iReset_Msg3235 -1,32767); END_IF		(* activate 'Message Hold Time' to avoid log clathering by repeated OpMsg entries *)
	xMsg3235.Reset 		:= 	iReset_Msg3235 < 1;		//.Reset := TRUE;
	xMsg3235();
	MM2VIS.bMsg3235		:=	xMsg3235.Q;

	xMsg3236.Enable		:=	IN_CU.tPB2MM.bParaSetupOk ;
	xMsg3236.Set		:=	OUT_CU.bMsg3236;		(* B3236 reserve operating message 5 *)
	IF xMsg3236.Set THEN iReset_Msg3236 := iDelay_MsgAutoReset_100ms; ELSE iReset_Msg3236 := LIMIT(0, iReset_Msg3236 -1,32767); END_IF		(* activate 'Message Hold Time' to avoid log clathering by repeated OpMsg entries *)
	xMsg3236.Reset 		:= 	iReset_Msg3236 < 1;		//.Reset := TRUE;
	xMsg3236();
	MM2VIS.bMsg3236		:=	xMsg3236.Q;

	xMsg3237.Enable		:=	IN_CU.tPB2MM.bParaSetupOk ;
	xMsg3237.Set		:=	OUT_CU.bMsg3237;		(* B3237 reserve operating message 6 *)
	IF xMsg3237.Set THEN iReset_Msg3237 := iDelay_MsgAutoReset_100ms; ELSE iReset_Msg3237 := LIMIT(0, iReset_Msg3237 -1,32767); END_IF		(* activate 'Message Hold Time' to avoid log clathering by repeated OpMsg entries *)
	xMsg3237.Reset 		:= 	iReset_Msg3237 < 1;		//.Reset := TRUE;
	xMsg3237();
	MM2VIS.bMsg3237		:=	xMsg3237.Q;
	(*----------------------------------------------------------------------*)

	xMsg3250.Enable		:=	IN_CU.tPB2MM.bParaSetupOk ;
	xMsg3250.Set		:=	OUT_CU.bMsg3250;		(* B3250 reserve operating message 7 *)
	IF xMsg3250.Set THEN iReset_Msg3250 := iDelay_MsgAutoReset_100ms; ELSE iReset_Msg3250 := LIMIT(0, iReset_Msg3250 -1,32767); END_IF		(* activate 'Message Hold Time' to avoid log clathering by repeated OpMsg entries *)
	xMsg3250.Reset 		:= 	iReset_Msg3250 < 1;		//.Reset := TRUE;
	xMsg3250();
	MM2VIS.bMsg3250		:=	xMsg3250.Q;

	xMsg3251.Enable		:=	IN_CU.tPB2MM.bParaSetupOk ;
	xMsg3251.Set		:=	OUT_CU.bMsg3251;		(* B3251 reserve operating message 8 *)
	IF xMsg3251.Set THEN iReset_Msg3251 := iDelay_MsgAutoReset_100ms; ELSE iReset_Msg3251 := LIMIT(0, iReset_Msg3251 -1,32767); END_IF		(* activate 'Message Hold Time' to avoid log clathering by repeated OpMsg entries *)
	xMsg3251.Reset 		:= 	iReset_Msg3251 < 1;		//.Reset := TRUE;
	xMsg3251();
	MM2VIS.bMsg3251		:=	xMsg3251.Q;
	(*----------------------------------------------------------------------*)

	xMsg36[01].Enable	:=	IN_CU.tPB2MM.bParaSetupOk ;
	xMsg36[01].Set		:=	OUT_CU.bMsg3601;		(* B3601 reserve operating message *)
	IF xMsg36[01].Set THEN iReset_Msg36[01] := iDelay_MsgAutoReset_100ms; ELSE iReset_Msg36[01] := LIMIT(0, iReset_Msg36[01] -1,32767); END_IF		(* activate 'Message Hold Time' to avoid log clathering by repeated OpMsg entries *)
	xMsg36[01].Reset	:= 	(iReset_Msg36[01] < 1);		//.Reset := TRUE;
	xMsg36[01]();
	MM2VIS.bMsg3601		:=	xMsg36[01].Q;

	xMsg36[02].Enable	:=	IN_CU.tPB2MM.bParaSetupOk ;
	xMsg36[02].Set		:=	OUT_CU.bMsg3602;			(* B3602 reserve operating message *)
	IF xMsg36[02].Set THEN iReset_Msg36[02] := iDelay_MsgAutoReset_100ms; ELSE iReset_Msg36[02] := LIMIT(0, iReset_Msg36[02] -1,32767); END_IF		(* activate 'Message Hold Time' to avoid log clathering by repeated OpMsg entries *)
	xMsg36[02].Reset 	:= 	(iReset_Msg36[02] < 1);		//.Reset := TRUE;
	xMsg36[02]();
	MM2VIS.bMsg3602		:=	xMsg36[02].Q;

	xMsg36[03].Enable	:=	IN_CU.tPB2MM.bParaSetupOk ;
	xMsg36[03].Set		:=	OUT_CU.bMsg3603;		(* B3603 reserve operating message *)
	IF xMsg36[03].Set THEN iReset_Msg36[03] := iDelay_MsgAutoReset_100ms; ELSE iReset_Msg36[03] := LIMIT(0, iReset_Msg36[03] -1,32767); END_IF		(* activate 'Message Hold Time' to avoid log clathering by repeated OpMsg entries *)
	xMsg36[03].Reset 	:= 	(iReset_Msg36[03] < 1);		//.Reset := TRUE;
	xMsg36[03]();
	MM2VIS.bMsg3603		:=	xMsg36[03].Q;

	xMsg36[04].Enable	:=	IN_CU.tPB2MM.bParaSetupOk ;
	xMsg36[04].Set		:=	OUT_CU.bMsg3604;		(* B3604 reserve operating message *)
	IF xMsg36[04].Set THEN iReset_Msg36[04] := iDelay_MsgAutoReset_100ms; ELSE iReset_Msg36[04] := LIMIT(0, iReset_Msg36[04] -1,32767); END_IF		(* activate 'Message Hold Time' to avoid log clathering by repeated OpMsg entries *)
	xMsg36[04].Reset 	:= 	(iReset_Msg36[04] < 1);		//.Reset := TRUE;
	xMsg36[04]();
	MM2VIS.bMsg3604		:=	xMsg36[04].Q;

	xMsg36[05].Enable	:=	IN_CU.tPB2MM.bParaSetupOk ;
	xMsg36[05].Set		:=	OUT_CU.bMsg3605;		(* B3605 reserve operating message *)
	IF xMsg36[05].Set THEN iReset_Msg36[05] := iDelay_MsgAutoReset_100ms; ELSE iReset_Msg36[05] := LIMIT(0, iReset_Msg36[05] -1,32767); END_IF		(* activate 'Message Hold Time' to avoid log clathering by repeated OpMsg entries *)
	xMsg36[05].Reset 	:= 	(iReset_Msg36[05] < 1);		//.Reset := TRUE;
	xMsg36[05]();
	MM2VIS.bMsg3605		:=	xMsg36[05].Q;

	xMsg36[06].Enable	:=	IN_CU.tPB2MM.bParaSetupOk ;
	xMsg36[06].Set		:=	OUT_CU.bMsg3606;		(* B3606 reserve operating message *)
	IF xMsg36[06].Set THEN iReset_Msg36[06] := iDelay_MsgAutoReset_100ms; ELSE iReset_Msg36[06] := LIMIT(0, iReset_Msg36[06] -1,32767); END_IF		(* activate 'Message Hold Time' to avoid log clathering by repeated OpMsg entries *)
	xMsg36[06].Reset 	:= 	(iReset_Msg36[06] < 1);		//.Reset := TRUE;
	xMsg36[06]();
	MM2VIS.bMsg3606		:=	xMsg36[06].Q;

	xMsg36[07].Enable	:=	IN_CU.tPB2MM.bParaSetupOk ;
	xMsg36[07].Set		:=	OUT_CU.bMsg3607;		(* B3607 reserve operating message *)
	IF xMsg36[07].Set THEN iReset_Msg36[07] := iDelay_MsgAutoReset_100ms; ELSE iReset_Msg36[07] := LIMIT(0, iReset_Msg36[07] -1,32767); END_IF		(* activate 'Message Hold Time' to avoid log clathering by repeated OpMsg entries *)
	xMsg36[07].Reset 	:= 	(iReset_Msg36[07] < 1);		//.Reset := TRUE;
	xMsg36[07]();
	MM2VIS.bMsg3607		:=	xMsg36[07].Q;

	xMsg36[08].Enable	:=	IN_CU.tPB2MM.bParaSetupOk ;
	xMsg36[08].Set		:=	OUT_CU.bMsg3608;		(* B3608 reserve operating message *)
	IF xMsg36[08].Set THEN iReset_Msg36[08] := iDelay_MsgAutoReset_100ms; ELSE iReset_Msg36[08] := LIMIT(0, iReset_Msg36[08] -1,32767); END_IF		(* activate 'Message Hold Time' to avoid log clathering by repeated OpMsg entries *)
	xMsg36[08].Reset 	:= 	(iReset_Msg36[08] < 1);		//.Reset := TRUE;
	xMsg36[08]();
	MM2VIS.bMsg3608		:=	xMsg36[08].Q;

	xMsg36[09].Enable	:=	IN_CU.tPB2MM.bParaSetupOk ;
	xMsg36[09].Set		:=	OUT_CU.bMsg3609;		(* B3609 reserve operating message *)
	IF xMsg36[09].Set THEN iReset_Msg36[09] := iDelay_MsgAutoReset_100ms; ELSE iReset_Msg36[09] := LIMIT(0, iReset_Msg36[09] -1,32767); END_IF		(* activate 'Message Hold Time' to avoid log clathering by repeated OpMsg entries *)
	xMsg36[09].Reset 	:= 	(iReset_Msg36[09] < 1);		//.Reset := TRUE;
	xMsg36[09]();
	MM2VIS.bMsg3609		:=	xMsg36[09].Q;

	xMsg36[10].Enable	:=	IN_CU.tPB2MM.bParaSetupOk ;
	xMsg36[10].Set		:=	OUT_CU.bMsg3610;		(* B3610 reserve operating message *)
	IF xMsg36[10].Set THEN iReset_Msg36[10] := iDelay_MsgAutoReset_100ms; ELSE iReset_Msg36[10] := LIMIT(0, iReset_Msg36[10] -1,32767); END_IF		(* activate 'Message Hold Time' to avoid log clathering by repeated OpMsg entries *)
	xMsg36[10].Reset 	:= 	(iReset_Msg36[10] < 1);		//.Reset := TRUE;
	xMsg36[10]();
	MM2VIS.bMsg3610		:=	xMsg36[10].Q;
	(*----------------------------------------------------------------------*)

	xMsg36[11].Enable	:=	IN_CU.tPB2MM.bParaSetupOk ;
	xMsg36[11].Set		:=	OUT_CU.bMsg3611;(* B3611 reserve operating message *)
	IF xMsg36[11].Set THEN iReset_Msg36[11] := iDelay_MsgAutoReset_100ms; ELSE iReset_Msg36[11] := LIMIT(0, iReset_Msg36[11] -1,32767); END_IF		(* activate 'Message Hold Time' to avoid log clathering by repeated OpMsg entries *)
	xMsg36[11].Reset 	:= 	(iReset_Msg36[11] < 1);		//.Reset := TRUE;
	xMsg36[11]();
	MM2VIS.bMsg3611		:=	xMsg36[11].Q;

	xMsg36[12].Enable	:=	IN_CU.tPB2MM.bParaSetupOk ;
	xMsg36[12].Set		:=	OUT_CU.bMsg3612;(* B3612 reserve operating message *)
	IF xMsg36[12].Set THEN iReset_Msg36[12] := iDelay_MsgAutoReset_100ms; ELSE iReset_Msg36[12] := LIMIT(0, iReset_Msg36[12] -1,32767); END_IF		(* activate 'Message Hold Time' to avoid log clathering by repeated OpMsg entries *)
	xMsg36[12].Reset 	:= 	(iReset_Msg36[12] < 1);		//.Reset := TRUE;
	xMsg36[12]();
	MM2VIS.bMsg3612		:=	xMsg36[12].Q;

	xMsg36[13].Enable	:=	IN_CU.tPB2MM.bParaSetupOk ;
	xMsg36[13].Set		:=	OUT_CU.bMsg3613;(* B3613 reserve operating message *)
	IF xMsg36[13].Set THEN iReset_Msg36[13] := iDelay_MsgAutoReset_100ms; ELSE iReset_Msg36[13] := LIMIT(0, iReset_Msg36[13] -1,32767); END_IF		(* activate 'Message Hold Time' to avoid log clathering by repeated OpMsg entries *)
	xMsg36[13].Reset 	:= 	(iReset_Msg36[13] < 1);		//.Reset := TRUE;
	xMsg36[13]();
	MM2VIS.bMsg3613		:=	xMsg36[13].Q;

	xMsg36[14].Enable	:=	IN_CU.tPB2MM.bParaSetupOk ;
	xMsg36[14].Set		:=	OUT_CU.bMsg3614;(* B3614 reserve operating message *)
	IF xMsg36[14].Set THEN iReset_Msg36[14] := iDelay_MsgAutoReset_100ms; ELSE iReset_Msg36[14] := LIMIT(0, iReset_Msg36[14] -1,32767); END_IF		(* activate 'Message Hold Time' to avoid log clathering by repeated OpMsg entries *)
	xMsg36[14].Reset 	:= 	(iReset_Msg36[14] < 1);		//.Reset := TRUE;
	xMsg36[14]();
	MM2VIS.bMsg3614		:=	xMsg36[14].Q;

	xMsg36[15].Enable	:=	IN_CU.tPB2MM.bParaSetupOk ;
	xMsg36[15].Set		:=	OUT_CU.bMsg3615;(* B3615 reserve operating message *)
	IF xMsg36[15].Set THEN iReset_Msg36[15] := iDelay_MsgAutoReset_100ms; ELSE iReset_Msg36[15] := LIMIT(0, iReset_Msg36[15] -1,32767); END_IF		(* activate 'Message Hold Time' to avoid log clathering by repeated OpMsg entries *)
	xMsg36[15].Reset 	:= 	(iReset_Msg36[15] < 1);		//.Reset := TRUE;
	xMsg36[15]();
	MM2VIS.bMsg3615		:=	xMsg36[15].Q;

	xMsg36[16].Enable	:=	IN_CU.tPB2MM.bParaSetupOk ;
	xMsg36[16].Set		:=	OUT_CU.bMsg3616;(* B3616 reserve operating message *)
	IF xMsg36[16].Set THEN iReset_Msg36[16] := iDelay_MsgAutoReset_100ms; ELSE iReset_Msg36[16] := LIMIT(0, iReset_Msg36[16] -1,32767); END_IF		(* activate 'Message Hold Time' to avoid log clathering by repeated OpMsg entries *)
	xMsg36[16].Reset 	:= 	(iReset_Msg36[16] < 1);		//.Reset := TRUE;
	xMsg36[16]();
	MM2VIS.bMsg3616		:=	xMsg36[16].Q;

	xMsg36[17].Enable	:=	IN_CU.tPB2MM.bParaSetupOk ;
	xMsg36[17].Set		:=	OUT_CU.bMsg3617;(* B3617 reserve operating message *)
	IF xMsg36[17].Set THEN iReset_Msg36[17] := iDelay_MsgAutoReset_100ms; ELSE iReset_Msg36[17] := LIMIT(0, iReset_Msg36[17] -1,32767); END_IF		(* activate 'Message Hold Time' to avoid log clathering by repeated OpMsg entries *)
	xMsg36[17].Reset 	:= 	(iReset_Msg36[17] < 1);		//.Reset := TRUE;
	xMsg36[17]();
	MM2VIS.bMsg3617		:=	xMsg36[17].Q;

	xMsg36[18].Enable	:=	IN_CU.tPB2MM.bParaSetupOk ;
	xMsg36[18].Set		:=	OUT_CU.bMsg3618;(* B3618 reserve operating message *)
	IF xMsg36[18].Set THEN iReset_Msg36[18] := iDelay_MsgAutoReset_100ms; ELSE iReset_Msg36[18] := LIMIT(0, iReset_Msg36[18] -1,32767); END_IF		(* activate 'Message Hold Time' to avoid log clathering by repeated OpMsg entries *)
	xMsg36[18].Reset 	:= 	(iReset_Msg36[18] < 1);		//.Reset := TRUE;
	xMsg36[18]();
	MM2VIS.bMsg3618		:=	xMsg36[18].Q;

	xMsg36[19].Enable	:=	IN_CU.tPB2MM.bParaSetupOk ;
	xMsg36[19].Set		:=	OUT_CU.bMsg3619;(* B3619 reserve operating message *)
	IF xMsg36[19].Set THEN iReset_Msg36[19] := iDelay_MsgAutoReset_100ms; ELSE iReset_Msg36[19] := LIMIT(0, iReset_Msg36[19] -1,32767); END_IF		(* activate 'Message Hold Time' to avoid log clathering by repeated OpMsg entries *)
	xMsg36[19].Reset 	:= 	(iReset_Msg36[19] < 1);		//.Reset := TRUE;
	xMsg36[19]();
	MM2VIS.bMsg3619		:=	xMsg36[19].Q;

	xMsg36[20].Enable	:=	IN_CU.tPB2MM.bParaSetupOk ;
	xMsg36[20].Set		:=	OUT_CU.bMsg3620;(* B3620 reserve operating message *)
	IF xMsg36[20].Set THEN iReset_Msg36[20] := iDelay_MsgAutoReset_100ms; ELSE iReset_Msg36[20] := LIMIT(0, iReset_Msg36[20] -1,32767); END_IF		(* activate 'Message Hold Time' to avoid log clathering by repeated OpMsg entries *)
	xMsg36[20].Reset 	:= 	(iReset_Msg36[20] < 1);		//.Reset := TRUE;
	xMsg36[20]();
	MM2VIS.bMsg3620		:=	xMsg36[20].Q;
	(*----------------------------------------------------------------------*)

	xMsg36[21].Enable	:=	IN_CU.tPB2MM.bParaSetupOk ;
	xMsg36[21].Set		:=	OUT_CU.bMsg3621;(* B3621 reserve operating message *)
	IF xMsg36[21].Set THEN iReset_Msg36[21] := iDelay_MsgAutoReset_100ms; ELSE iReset_Msg36[21] := LIMIT(0, iReset_Msg36[21] -1,32767); END_IF		(* activate 'Message Hold Time' to avoid log clathering by repeated OpMsg entries *)
	xMsg36[21].Reset 	:= 	(iReset_Msg36[21] < 1);		//.Reset := TRUE;
	xMsg36[21]();
	MM2VIS.bMsg3621		:=	xMsg36[21].Q;

	xMsg36[22].Enable	:=	IN_CU.tPB2MM.bParaSetupOk ;
	xMsg36[22].Set		:=	OUT_CU.bMsg3622;(* B3622 reserve operating message *)
	IF xMsg36[22].Set THEN iReset_Msg36[22] := iDelay_MsgAutoReset_100ms; ELSE iReset_Msg36[22] := LIMIT(0, iReset_Msg36[22] -1,32767); END_IF		(* activate 'Message Hold Time' to avoid log clathering by repeated OpMsg entries *)
	xMsg36[22].Reset 	:= 	(iReset_Msg36[22] < 1);		//.Reset := TRUE;
	xMsg36[22]();
	MM2VIS.bMsg3622		:=	xMsg36[22].Q;

	xMsg36[23].Enable	:=	IN_CU.tPB2MM.bParaSetupOk ;
	xMsg36[23].Set		:=	OUT_CU.bMsg3623;(* B3623 reserve operating message *)
	IF xMsg36[23].Set THEN iReset_Msg36[23] := iDelay_MsgAutoReset_100ms; ELSE iReset_Msg36[23] := LIMIT(0, iReset_Msg36[23] -1,32767); END_IF		(* activate 'Message Hold Time' to avoid log clathering by repeated OpMsg entries *)
	xMsg36[23].Reset 	:= 	(iReset_Msg36[23] < 1);		//.Reset := TRUE;
	xMsg36[23]();
	MM2VIS.bMsg3623		:=	xMsg36[23].Q;

	xMsg36[24].Enable	:=	IN_CU.tPB2MM.bParaSetupOk ;
	xMsg36[24].Set		:=	OUT_CU.bMsg3624;(* B3624 reserve operating message *)
	IF xMsg36[24].Set THEN iReset_Msg36[24] := iDelay_MsgAutoReset_100ms; ELSE iReset_Msg36[24] := LIMIT(0, iReset_Msg36[24] -1,32767); END_IF		(* activate 'Message Hold Time' to avoid log clathering by repeated OpMsg entries *)
	xMsg36[24].Reset 	:= 	(iReset_Msg36[24] < 1);		//.Reset := TRUE;
	xMsg36[24]();
	MM2VIS.bMsg3624		:=	xMsg36[24].Q;

	xMsg36[25].Enable	:=	IN_CU.tPB2MM.bParaSetupOk ;
	xMsg36[25].Set		:=	OUT_CU.bMsg3625;(* B3625 reserve operating message *)
	IF xMsg36[25].Set THEN iReset_Msg36[25] := iDelay_MsgAutoReset_100ms; ELSE iReset_Msg36[25] := LIMIT(0, iReset_Msg36[25] -1,32767); END_IF		(* activate 'Message Hold Time' to avoid log clathering by repeated OpMsg entries *)
	xMsg36[25].Reset 	:= 	(iReset_Msg36[25] < 1);		//.Reset := TRUE;
	xMsg36[25]();
	MM2VIS.bMsg3625		:=	xMsg36[25].Q;

	xMsg36[26].Enable	:=	IN_CU.tPB2MM.bParaSetupOk ;
	xMsg36[26].Set		:=	OUT_CU.bMsg3626;(* B3626 reserve operating message *)
	IF xMsg36[26].Set THEN iReset_Msg36[26] := iDelay_MsgAutoReset_100ms; ELSE iReset_Msg36[26] := LIMIT(0, iReset_Msg36[26] -1,32767); END_IF		(* activate 'Message Hold Time' to avoid log clathering by repeated OpMsg entries *)
	xMsg36[26].Reset 	:= 	(iReset_Msg36[26] < 1);		//.Reset := TRUE;
	xMsg36[26]();
	MM2VIS.bMsg3626		:=	xMsg36[26].Q;

	xMsg36[27].Enable	:=	IN_CU.tPB2MM.bParaSetupOk ;
	xMsg36[27].Set		:=	OUT_CU.bMsg3627;(* B3627 reserve operating message *)
	IF xMsg36[27].Set THEN iReset_Msg36[27] := iDelay_MsgAutoReset_100ms; ELSE iReset_Msg36[27] := LIMIT(0, iReset_Msg36[27] -1,32767); END_IF		(* activate 'Message Hold Time' to avoid log clathering by repeated OpMsg entries *)
	xMsg36[27].Reset 	:= 	(iReset_Msg36[27] < 1);		//.Reset := TRUE;
	xMsg36[27]();
	MM2VIS.bMsg3627		:=	xMsg36[27].Q;

	xMsg36[28].Enable	:=	IN_CU.tPB2MM.bParaSetupOk ;
	xMsg36[28].Set		:=	OUT_CU.bMsg3628;(* B3628 reserve operating message *)
	IF xMsg36[28].Set THEN iReset_Msg36[28] := iDelay_MsgAutoReset_100ms; ELSE iReset_Msg36[28] := LIMIT(0, iReset_Msg36[28] -1,32767); END_IF		(* activate 'Message Hold Time' to avoid log clathering by repeated OpMsg entries *)
	xMsg36[28].Reset 	:= 	(iReset_Msg36[28] < 1);		//.Reset := TRUE;
	xMsg36[28]();
	MM2VIS.bMsg3628		:=	xMsg36[28].Q;

	xMsg36[29].Enable	:=	IN_CU.tPB2MM.bParaSetupOk ;
	xMsg36[29].Set		:=	OUT_CU.bMsg3629;(* B3629 reserve operating message *)
	IF xMsg36[29].Set THEN iReset_Msg36[29] := iDelay_MsgAutoReset_100ms; ELSE iReset_Msg36[29] := LIMIT(0, iReset_Msg36[29] -1,32767); END_IF		(* activate 'Message Hold Time' to avoid log clathering by repeated OpMsg entries *)
	xMsg36[29].Reset 	:= 	(iReset_Msg36[29] < 1);		//.Reset := TRUE;
	xMsg36[29]();
	MM2VIS.bMsg3629		:=	xMsg36[29].Q;

	xMsg36[30].Enable	:=	IN_CU.tPB2MM.bParaSetupOk ;
	xMsg36[30].Set		:=	OUT_CU.bMsg3630;(* B3630 reserve operating message *)
	IF xMsg36[30].Set THEN iReset_Msg36[30] := iDelay_MsgAutoReset_100ms; ELSE iReset_Msg36[30] := LIMIT(0, iReset_Msg36[30] -1,32767); END_IF		(* activate 'Message Hold Time' to avoid log clathering by repeated OpMsg entries *)
	xMsg36[30].Reset 	:= 	(iReset_Msg36[30] < 1);		//.Reset := TRUE;
	xMsg36[30]();
	MM2VIS.bMsg3630		:=	xMsg36[30].Q;
	(*----------------------------------------------------------------------*)

	xMsg36[31].Enable	:=	IN_CU.tPB2MM.bParaSetupOk ;
	xMsg36[31].Set		:=	OUT_CU.bMsg3631;(* B3631 reserve operating message *)
	IF xMsg36[31].Set THEN iReset_Msg36[31] := iDelay_MsgAutoReset_100ms; ELSE iReset_Msg36[31] := LIMIT(0, iReset_Msg36[31] -1,32767); END_IF		(* activate 'Message Hold Time' to avoid log clathering by repeated OpMsg entries *)
	xMsg36[31].Reset 	:= 	(iReset_Msg36[31] < 1);		//.Reset := TRUE;
	xMsg36[31]();
	MM2VIS.bMsg3631		:=	xMsg36[31].Q;

	xMsg36[32].Enable	:=	IN_CU.tPB2MM.bParaSetupOk ;
	xMsg36[32].Set		:=	OUT_CU.bMsg3632;(* B3632 reserve operating message *)
	IF xMsg36[32].Set THEN iReset_Msg36[32] := iDelay_MsgAutoReset_100ms; ELSE iReset_Msg36[32] := LIMIT(0, iReset_Msg36[32] -1,32767); END_IF		(* activate 'Message Hold Time' to avoid log clathering by repeated OpMsg entries *)
	xMsg36[32].Reset 	:= 	(iReset_Msg36[32] < 1);		//.Reset := TRUE;
	xMsg36[32]();
	MM2VIS.bMsg3632		:=	xMsg36[32].Q;

	xMsg36[33].Enable	:=	IN_CU.tPB2MM.bParaSetupOk ;
	xMsg36[33].Set		:=	OUT_CU.bMsg3633;(* B3633 reserve operating message *)
	IF xMsg36[33].Set THEN iReset_Msg36[33] := iDelay_MsgAutoReset_100ms; ELSE iReset_Msg36[33] := LIMIT(0, iReset_Msg36[33] -1,32767); END_IF		(* activate 'Message Hold Time' to avoid log clathering by repeated OpMsg entries *)
	xMsg36[33].Reset 	:= 	(iReset_Msg36[33] < 1);		//.Reset := TRUE;
	xMsg36[33]();
	MM2VIS.bMsg3633		:=	xMsg36[33].Q;

	xMsg36[34].Enable	:=	IN_CU.tPB2MM.bParaSetupOk ;
	xMsg36[34].Set		:=	OUT_CU.bMsg3634;(* B3634 reserve operating message *)
	IF xMsg36[34].Set THEN iReset_Msg36[34] := iDelay_MsgAutoReset_100ms; ELSE iReset_Msg36[34] := LIMIT(0, iReset_Msg36[34] -1,32767); END_IF		(* activate 'Message Hold Time' to avoid log clathering by repeated OpMsg entries *)
	xMsg36[34].Reset 	:= 	(iReset_Msg36[34] < 1);		//.Reset := TRUE;
	xMsg36[34]();
	MM2VIS.bMsg3634		:=	xMsg36[34].Q;

	xMsg36[35].Enable	:=	IN_CU.tPB2MM.bParaSetupOk ;
	xMsg36[35].Set		:=	OUT_CU.bMsg3635;(* B3635 reserve operating message *)
	IF xMsg36[35].Set THEN iReset_Msg36[35] := iDelay_MsgAutoReset_100ms; ELSE iReset_Msg36[35] := LIMIT(0, iReset_Msg36[35] -1,32767); END_IF		(* activate 'Message Hold Time' to avoid log clathering by repeated OpMsg entries *)
	xMsg36[35].Reset 	:= 	(iReset_Msg36[35] < 1);		//.Reset := TRUE;
	xMsg36[35]();
	MM2VIS.bMsg3635		:=	xMsg36[35].Q;

	xMsg36[36].Enable	:=	IN_CU.tPB2MM.bParaSetupOk ;
	xMsg36[36].Set		:=	OUT_CU.bMsg3636;(* B3636 reserve operating message *)
	IF xMsg36[36].Set THEN iReset_Msg36[36] := iDelay_MsgAutoReset_100ms; ELSE iReset_Msg36[36] := LIMIT(0, iReset_Msg36[36] -1,32767); END_IF		(* activate 'Message Hold Time' to avoid log clathering by repeated OpMsg entries *)
	xMsg36[36].Reset 	:= 	(iReset_Msg36[36] < 1);		//.Reset := TRUE;
	xMsg36[36]();
	MM2VIS.bMsg3636		:=	xMsg36[36].Q;

	xMsg36[37].Enable	:=	IN_CU.tPB2MM.bParaSetupOk ;
	xMsg36[37].Set		:=	OUT_CU.bMsg3637;(* B3637 reserve operating message *)
	IF xMsg36[37].Set THEN iReset_Msg36[37] := iDelay_MsgAutoReset_100ms; ELSE iReset_Msg36[37] := LIMIT(0, iReset_Msg36[37] -1,32767); END_IF		(* activate 'Message Hold Time' to avoid log clathering by repeated OpMsg entries *)
	xMsg36[37].Reset 	:= 	(iReset_Msg36[37] < 1);		//.Reset := TRUE;
	xMsg36[37]();
	MM2VIS.bMsg3637		:=	xMsg36[37].Q;

	xMsg36[38].Enable	:=	IN_CU.tPB2MM.bParaSetupOk ;
	xMsg36[38].Set		:=	OUT_CU.bMsg3638;(* B3638 reserve operating message *)
	IF xMsg36[38].Set THEN iReset_Msg36[38] := iDelay_MsgAutoReset_100ms; ELSE iReset_Msg36[38] := LIMIT(0, iReset_Msg36[38] -1,32767); END_IF		(* activate 'Message Hold Time' to avoid log clathering by repeated OpMsg entries *)
	xMsg36[38].Reset 	:= 	(iReset_Msg36[38] < 1);		//.Reset := TRUE;
	xMsg36[38]();
	MM2VIS.bMsg3638		:=	xMsg36[38].Q;

	xMsg36[39].Enable	:=	IN_CU.tPB2MM.bParaSetupOk ;
	xMsg36[39].Set		:=	OUT_CU.bMsg3639;(* B3639 reserve operating message *)
	IF xMsg36[39].Set THEN iReset_Msg36[39] := iDelay_MsgAutoReset_100ms; ELSE iReset_Msg36[39] := LIMIT(0, iReset_Msg36[39] -1,32767); END_IF		(* activate 'Message Hold Time' to avoid log clathering by repeated OpMsg entries *)
	xMsg36[39].Reset 	:= 	(iReset_Msg36[39] < 1);		//.Reset := TRUE;
	xMsg36[39]();
	MM2VIS.bMsg3639		:=	xMsg36[39].Q;

	xMsg36[40].Enable	:=	IN_CU.tPB2MM.bParaSetupOk ;
	xMsg36[40].Set		:=	OUT_CU.bMsg3640;(* B3640 reserve operating message *)
	IF xMsg36[40].Set THEN iReset_Msg36[40] := iDelay_MsgAutoReset_100ms; ELSE iReset_Msg36[40] := LIMIT(0, iReset_Msg36[40] -1,32767); END_IF		(* activate 'Message Hold Time' to avoid log clathering by repeated OpMsg entries *)
	xMsg36[40].Reset 	:= 	(iReset_Msg36[40] < 1);		//.Reset := TRUE;
	xMsg36[40]();
	MM2VIS.bMsg3640		:=	xMsg36[40].Q;
	(*----------------------------------------------------------------------*)

	xMsg36[41].Enable	:=	IN_CU.tPB2MM.bParaSetupOk ;
	xMsg36[41].Set		:=	OUT_CU.bMsg3641;(* B3641 reserve operating message *)
	IF xMsg36[41].Set THEN iReset_Msg36[41] := iDelay_MsgAutoReset_100ms; ELSE iReset_Msg36[41] := LIMIT(0, iReset_Msg36[41] -1,32767); END_IF		(* activate 'Message Hold Time' to avoid log clathering by repeated OpMsg entries *)
	xMsg36[41].Reset 	:= 	(iReset_Msg36[41] < 1);		//.Reset := TRUE;
	xMsg36[41]();
	MM2VIS.bMsg3641		:=	xMsg36[41].Q;

	xMsg36[42].Enable	:=	IN_CU.tPB2MM.bParaSetupOk ;
	xMsg36[42].Set		:=	OUT_CU.bMsg3642;(* B3642 reserve operating message *)
	IF xMsg36[42].Set THEN iReset_Msg36[42] := iDelay_MsgAutoReset_100ms; ELSE iReset_Msg36[42] := LIMIT(0, iReset_Msg36[42] -1,32767); END_IF		(* activate 'Message Hold Time' to avoid log clathering by repeated OpMsg entries *)
	xMsg36[42].Reset 	:= 	(iReset_Msg36[42] < 1);		//.Reset := TRUE;
	xMsg36[42]();
	MM2VIS.bMsg3642		:=	xMsg36[42].Q;

	xMsg36[43].Enable	:=	IN_CU.tPB2MM.bParaSetupOk ;
	xMsg36[43].Set		:=	OUT_CU.bMsg3643;(* B3643 reserve operating message *)
	IF xMsg36[43].Set THEN iReset_Msg36[43] := iDelay_MsgAutoReset_100ms; ELSE iReset_Msg36[43] := LIMIT(0, iReset_Msg36[43] -1,32767); END_IF		(* activate 'Message Hold Time' to avoid log clathering by repeated OpMsg entries *)
	xMsg36[43].Reset 	:= 	(iReset_Msg36[43] < 1);		//.Reset := TRUE;
	xMsg36[43]();
	MM2VIS.bMsg3643		:=	xMsg36[43].Q;

	xMsg36[44].Enable	:=	IN_CU.tPB2MM.bParaSetupOk ;
	xMsg36[44].Set		:=	OUT_CU.bMsg3644;(* B3644 reserve operating message *)
	IF xMsg36[44].Set THEN iReset_Msg36[44] := iDelay_MsgAutoReset_100ms; ELSE iReset_Msg36[44] := LIMIT(0, iReset_Msg36[44] -1,32767); END_IF		(* activate 'Message Hold Time' to avoid log clathering by repeated OpMsg entries *)
	xMsg36[44].Reset 	:= 	(iReset_Msg36[44] < 1);		//.Reset := TRUE;
	xMsg36[44]();
	MM2VIS.bMsg3644		:=	xMsg36[44].Q;

	xMsg36[45].Enable	:=	IN_CU.tPB2MM.bParaSetupOk ;
	xMsg36[45].Set		:=	OUT_CU.bMsg3645;(* B3645 reserve operating message *)
	IF xMsg36[45].Set THEN iReset_Msg36[45] := iDelay_MsgAutoReset_100ms; ELSE iReset_Msg36[45] := LIMIT(0, iReset_Msg36[45] -1,32767); END_IF		(* activate 'Message Hold Time' to avoid log clathering by repeated OpMsg entries *)
	xMsg36[45].Reset 	:= 	(iReset_Msg36[45] < 1);		//.Reset := TRUE;
	xMsg36[45]();
	MM2VIS.bMsg3645		:=	xMsg36[45].Q;

	xMsg36[46].Enable	:=	IN_CU.tPB2MM.bParaSetupOk ;
	xMsg36[46].Set		:=	OUT_CU.bMsg3646;(* B3646 reserve operating message *)
	IF xMsg36[46].Set THEN iReset_Msg36[46] := iDelay_MsgAutoReset_100ms; ELSE iReset_Msg36[46] := LIMIT(0, iReset_Msg36[46] -1,32767); END_IF		(* activate 'Message Hold Time' to avoid log clathering by repeated OpMsg entries *)
	xMsg36[46].Reset 	:= 	(iReset_Msg36[46] < 1);		//.Reset := TRUE;
	xMsg36[46]();
	MM2VIS.bMsg3646		:=	xMsg36[46].Q;

	xMsg36[47].Enable	:=	IN_CU.tPB2MM.bParaSetupOk ;
	xMsg36[47].Set		:=	OUT_CU.bMsg3647;(* B3647 reserve operating message *)
	IF xMsg36[47].Set THEN iReset_Msg36[47] := iDelay_MsgAutoReset_100ms; ELSE iReset_Msg36[47] := LIMIT(0, iReset_Msg36[47] -1,32767); END_IF		(* activate 'Message Hold Time' to avoid log clathering by repeated OpMsg entries *)
	xMsg36[47].Reset 	:= 	(iReset_Msg36[47] < 1);		//.Reset := TRUE;
	xMsg36[47]();
	MM2VIS.bMsg3647		:=	xMsg36[47].Q;

	xMsg36[48].Enable	:=	IN_CU.tPB2MM.bParaSetupOk ;
	xMsg36[48].Set		:=	OUT_CU.bMsg3648;(* B3648 reserve operating message *)
	IF xMsg36[48].Set THEN iReset_Msg36[48] := iDelay_MsgAutoReset_100ms; ELSE iReset_Msg36[48] := LIMIT(0, iReset_Msg36[48] -1,32767); END_IF		(* activate 'Message Hold Time' to avoid log clathering by repeated OpMsg entries *)
	xMsg36[48].Reset 	:= 	(iReset_Msg36[48] < 1);		//.Reset := TRUE;
	xMsg36[48]();
	MM2VIS.bMsg3648		:=	xMsg36[48].Q;

	xMsg36[49].Enable	:=	IN_CU.tPB2MM.bParaSetupOk ;
	xMsg36[49].Set		:=	OUT_CU.bMsg3649;(* B3649 reserve operating message *)
	IF xMsg36[49].Set THEN iReset_Msg36[49] := iDelay_MsgAutoReset_100ms; ELSE iReset_Msg36[49] := LIMIT(0, iReset_Msg36[49] -1,32767); END_IF		(* activate 'Message Hold Time' to avoid log clathering by repeated OpMsg entries *)
	xMsg36[49].Reset 	:= 	(iReset_Msg36[49] < 1);		//.Reset := TRUE;
	xMsg36[49]();
	MM2VIS.bMsg3649		:=	xMsg36[49].Q;

	xMsg36[50].Enable	:=	IN_CU.tPB2MM.bParaSetupOk ;
	xMsg36[50].Set		:=	OUT_CU.bMsg3650;(* B3650 reserve operating message *)
	IF xMsg36[50].Set THEN iReset_Msg36[50] := iDelay_MsgAutoReset_100ms; ELSE iReset_Msg36[50] := LIMIT(0, iReset_Msg36[50] -1,32767); END_IF		(* activate 'Message Hold Time' to avoid log clathering by repeated OpMsg entries *)
	xMsg36[50].Reset 	:= 	(iReset_Msg36[50] < 1);		//.Reset := TRUE;
	xMsg36[50]();
	MM2VIS.bMsg3650		:=	xMsg36[50].Q;
	(*----------------------------------------------------------------------*)

	xMsg36[51].Enable	:=	IN_CU.tPB2MM.bParaSetupOk ;
	xMsg36[51].Set		:=	OUT_CU.bMsg3651;(* B3651 reserve operating message *)
	IF xMsg36[51].Set THEN iReset_Msg36[51] := iDelay_MsgAutoReset_100ms; ELSE iReset_Msg36[51] := LIMIT(0, iReset_Msg36[51] -1,32767); END_IF		(* activate 'Message Hold Time' to avoid log clathering by repeated OpMsg entries *)
	xMsg36[51].Reset 	:= 	(iReset_Msg36[51] < 1);		//.Reset := TRUE;
	xMsg36[51]();
	MM2VIS.bMsg3651		:=	xMsg36[51].Q;

	xMsg36[52].Enable	:=	IN_CU.tPB2MM.bParaSetupOk ;
	xMsg36[52].Set		:=	OUT_CU.bMsg3652;(* B3652 reserve operating message *)
	IF xMsg36[52].Set THEN iReset_Msg36[52] := iDelay_MsgAutoReset_100ms; ELSE iReset_Msg36[52] := LIMIT(0, iReset_Msg36[52] -1,32767); END_IF		(* activate 'Message Hold Time' to avoid log clathering by repeated OpMsg entries *)
	xMsg36[52].Reset 	:= 	(iReset_Msg36[52] < 1);		//.Reset := TRUE;
	xMsg36[52]();
	MM2VIS.bMsg3652		:=	xMsg36[52].Q;

	xMsg36[53].Enable	:=	IN_CU.tPB2MM.bParaSetupOk ;
	xMsg36[53].Set		:=	OUT_CU.bMsg3653;(* B3653 reserve operating message *)
	IF xMsg36[53].Set THEN iReset_Msg36[53] := iDelay_MsgAutoReset_100ms; ELSE iReset_Msg36[53] := LIMIT(0, iReset_Msg36[53] -1,32767); END_IF		(* activate 'Message Hold Time' to avoid log clathering by repeated OpMsg entries *)
	xMsg36[53].Reset 	:= 	(iReset_Msg36[53] < 1);		//.Reset := TRUE;
	xMsg36[53]();
	MM2VIS.bMsg3653		:=	xMsg36[53].Q;

	xMsg36[54].Enable	:=	IN_CU.tPB2MM.bParaSetupOk ;
	xMsg36[54].Set		:=	OUT_CU.bMsg3654;(* B3654 reserve operating message *)
	IF xMsg36[54].Set THEN iReset_Msg36[54] := iDelay_MsgAutoReset_100ms; ELSE iReset_Msg36[54] := LIMIT(0, iReset_Msg36[54] -1,32767); END_IF		(* activate 'Message Hold Time' to avoid log clathering by repeated OpMsg entries *)
	xMsg36[54].Reset 	:= 	(iReset_Msg36[54] < 1);		//.Reset := TRUE;
	xMsg36[54]();
	MM2VIS.bMsg3654		:=	xMsg36[54].Q;

	xMsg36[55].Enable	:=	IN_CU.tPB2MM.bParaSetupOk ;
	xMsg36[55].Set		:=	OUT_CU.bMsg3655;(* B3655 reserve operating message *)
	IF xMsg36[55].Set THEN iReset_Msg36[55] := iDelay_MsgAutoReset_100ms; ELSE iReset_Msg36[55] := LIMIT(0, iReset_Msg36[55] -1,32767); END_IF		(* activate 'Message Hold Time' to avoid log clathering by repeated OpMsg entries *)
	xMsg36[55].Reset 	:= 	(iReset_Msg36[55] < 1);		//.Reset := TRUE;
	xMsg36[55]();
	MM2VIS.bMsg3655		:=	xMsg36[55].Q;

	xMsg36[56].Enable	:=	IN_CU.tPB2MM.bParaSetupOk ;
	xMsg36[56].Set		:=	OUT_CU.bMsg3656;(* B3656 reserve operating message *)
	IF xMsg36[56].Set THEN iReset_Msg36[56] := iDelay_MsgAutoReset_100ms; ELSE iReset_Msg36[56] := LIMIT(0, iReset_Msg36[56] -1,32767); END_IF		(* activate 'Message Hold Time' to avoid log clathering by repeated OpMsg entries *)
	xMsg36[56].Reset 	:= 	(iReset_Msg36[56] < 1);		//.Reset := TRUE;
	xMsg36[56]();
	MM2VIS.bMsg3656		:=	xMsg36[56].Q;

	xMsg36[57].Enable	:=	IN_CU.tPB2MM.bParaSetupOk ;
	xMsg36[57].Set		:=	OUT_CU.bMsg3657;(* B3657 reserve operating message *)
	IF xMsg36[57].Set THEN iReset_Msg36[57] := iDelay_MsgAutoReset_100ms; ELSE iReset_Msg36[57] := LIMIT(0, iReset_Msg36[57] -1,32767); END_IF		(* activate 'Message Hold Time' to avoid log clathering by repeated OpMsg entries *)
	xMsg36[57].Reset 	:= 	(iReset_Msg36[57] < 1);		//.Reset := TRUE;
	xMsg36[57]();
	MM2VIS.bMsg3657		:=	xMsg36[57].Q;

	xMsg36[58].Enable	:=	IN_CU.tPB2MM.bParaSetupOk ;
	xMsg36[58].Set		:=	OUT_CU.bMsg3658;(* B3658 reserve operating message *)
	IF xMsg36[58].Set THEN iReset_Msg36[58] := iDelay_MsgAutoReset_100ms; ELSE iReset_Msg36[58] := LIMIT(0, iReset_Msg36[58] -1,32767); END_IF		(* activate 'Message Hold Time' to avoid log clathering by repeated OpMsg entries *)
	xMsg36[58].Reset 	:= 	(iReset_Msg36[58] < 1);		//.Reset := TRUE;
	xMsg36[58]();
	MM2VIS.bMsg3658		:=	xMsg36[58].Q;

	xMsg36[59].Enable	:=	IN_CU.tPB2MM.bParaSetupOk ;
	xMsg36[59].Set		:=	OUT_CU.bMsg3659;(* B3659 reserve operating message *)
	IF xMsg36[59].Set THEN iReset_Msg36[59] := iDelay_MsgAutoReset_100ms; ELSE iReset_Msg36[59] := LIMIT(0, iReset_Msg36[59] -1,32767); END_IF		(* activate 'Message Hold Time' to avoid log clathering by repeated OpMsg entries *)
	xMsg36[59].Reset 	:= 	(iReset_Msg36[59] < 1);		//.Reset := TRUE;
	xMsg36[59]();
	MM2VIS.bMsg3659		:=	xMsg36[59].Q;

	xMsg36[60].Enable	:=	IN_CU.tPB2MM.bParaSetupOk ;
	xMsg36[60].Set		:=	OUT_CU.bMsg3660;(* B3660 reserve operating message *)
	IF xMsg36[60].Set THEN iReset_Msg36[60] := iDelay_MsgAutoReset_100ms; ELSE iReset_Msg36[60] := LIMIT(0, iReset_Msg36[60] -1,32767); END_IF		(* activate 'Message Hold Time' to avoid log clathering by repeated OpMsg entries *)
	xMsg36[60].Reset 	:= 	(iReset_Msg36[60] < 1);		//.Reset := TRUE;
	xMsg36[60]();
	MM2VIS.bMsg3660		:=	xMsg36[60].Q;
	(*----------------------------------------------------------------------*)

	xMsg36[61].Enable	:=	IN_CU.tPB2MM.bParaSetupOk ;
	xMsg36[61].Set		:=	OUT_CU.bMsg3661;(* B3661 reserve operating message *)
	IF xMsg36[61].Set THEN iReset_Msg36[61] := iDelay_MsgAutoReset_100ms; ELSE iReset_Msg36[61] := LIMIT(0, iReset_Msg36[61] -1,32767); END_IF		(* activate 'Message Hold Time' to avoid log clathering by repeated OpMsg entries *)
	xMsg36[61].Reset 	:= 	(iReset_Msg36[61] < 1);		//.Reset := TRUE;
	xMsg36[61]();
	MM2VIS.bMsg3661		:=	xMsg36[61].Q;

	xMsg36[62].Enable	:=	IN_CU.tPB2MM.bParaSetupOk ;
	xMsg36[62].Set		:=	OUT_CU.bMsg3662;(* B3662 reserve operating message *)
	IF xMsg36[62].Set THEN iReset_Msg36[62] := iDelay_MsgAutoReset_100ms; ELSE iReset_Msg36[62] := LIMIT(0, iReset_Msg36[62] -1,32767); END_IF		(* activate 'Message Hold Time' to avoid log clathering by repeated OpMsg entries *)
	xMsg36[62].Reset 	:= 	(iReset_Msg36[62] < 1);		//.Reset := TRUE;
	xMsg36[62]();
	MM2VIS.bMsg3662		:=	xMsg36[62].Q;

	xMsg36[63].Enable	:=	IN_CU.tPB2MM.bParaSetupOk ;
	xMsg36[63].Set		:=	OUT_CU.bMsg3663;(* B3663 reserve operating message *)
	IF xMsg36[63].Set THEN iReset_Msg36[63] := iDelay_MsgAutoReset_100ms; ELSE iReset_Msg36[63] := LIMIT(0, iReset_Msg36[63] -1,32767); END_IF		(* activate 'Message Hold Time' to avoid log clathering by repeated OpMsg entries *)
	xMsg36[63].Reset 	:= 	(iReset_Msg36[63] < 1);		//.Reset := TRUE;
	xMsg36[63]();
	MM2VIS.bMsg3663		:=	xMsg36[63].Q;

	xMsg36[64].Enable	:=	IN_CU.tPB2MM.bParaSetupOk ;
	xMsg36[64].Set		:=	OUT_CU.bMsg3664;(* B3664 reserve operating message *)
	IF xMsg36[64].Set THEN iReset_Msg36[64] := iDelay_MsgAutoReset_100ms; ELSE iReset_Msg36[64] := LIMIT(0, iReset_Msg36[64] -1,32767); END_IF		(* activate 'Message Hold Time' to avoid log clathering by repeated OpMsg entries *)
	xMsg36[64].Reset 	:= 	(iReset_Msg36[64] < 1);		//.Reset := TRUE;
	xMsg36[64]();
	MM2VIS.bMsg3664		:=	xMsg36[64].Q;

	xMsg36[65].Enable	:=	IN_CU.tPB2MM.bParaSetupOk ;
	xMsg36[65].Set		:=	OUT_CU.bMsg3665;(* B3665 reserve operating message *)
	IF xMsg36[65].Set THEN iReset_Msg36[65] := iDelay_MsgAutoReset_100ms; ELSE iReset_Msg36[65] := LIMIT(0, iReset_Msg36[65] -1,32767); END_IF		(* activate 'Message Hold Time' to avoid log clathering by repeated OpMsg entries *)
	xMsg36[65].Reset 	:= 	(iReset_Msg36[65] < 1);		//.Reset := TRUE;
	xMsg36[65]();
	MM2VIS.bMsg3665		:=	xMsg36[65].Q;

	xMsg36[66].Enable	:=	IN_CU.tPB2MM.bParaSetupOk ;
	xMsg36[66].Set		:=	OUT_CU.bMsg3666;(* B3666 reserve operating message *)
	IF xMsg36[66].Set THEN iReset_Msg36[66] := iDelay_MsgAutoReset_100ms; ELSE iReset_Msg36[66] := LIMIT(0, iReset_Msg36[66] -1,32767); END_IF		(* activate 'Message Hold Time' to avoid log clathering by repeated OpMsg entries *)
	xMsg36[66].Reset 	:= 	(iReset_Msg36[66] < 1);		//.Reset := TRUE;
	xMsg36[66]();
	MM2VIS.bMsg3666		:=	xMsg36[66].Q;

	xMsg36[67].Enable	:=	IN_CU.tPB2MM.bParaSetupOk ;
	xMsg36[67].Set		:=	OUT_CU.bMsg3667;(* B3667 reserve operating message *)
	IF xMsg36[67].Set THEN iReset_Msg36[67] := iDelay_MsgAutoReset_100ms; ELSE iReset_Msg36[67] := LIMIT(0, iReset_Msg36[67] -1,32767); END_IF		(* activate 'Message Hold Time' to avoid log clathering by repeated OpMsg entries *)
	xMsg36[67].Reset 	:= 	(iReset_Msg36[67] < 1);		//.Reset := TRUE;
	xMsg36[67]();
	MM2VIS.bMsg3667		:=	xMsg36[67].Q;

	xMsg36[68].Enable	:=	IN_CU.tPB2MM.bParaSetupOk ;
	xMsg36[68].Set		:=	OUT_CU.bMsg3668;(* B3668 reserve operating message *)
	IF xMsg36[68].Set THEN iReset_Msg36[68] := iDelay_MsgAutoReset_100ms; ELSE iReset_Msg36[68] := LIMIT(0, iReset_Msg36[68] -1,32767); END_IF		(* activate 'Message Hold Time' to avoid log clathering by repeated OpMsg entries *)
	xMsg36[68].Reset 	:= 	(iReset_Msg36[68] < 1);		//.Reset := TRUE;
	xMsg36[68]();
	MM2VIS.bMsg3668		:=	xMsg36[68].Q;

	xMsg36[69].Enable	:=	IN_CU.tPB2MM.bParaSetupOk ;
	xMsg36[69].Set		:=	OUT_CU.bMsg3669;(* B3669 reserve operating message *)
	IF xMsg36[69].Set THEN iReset_Msg36[69] := iDelay_MsgAutoReset_100ms; ELSE iReset_Msg36[69] := LIMIT(0, iReset_Msg36[69] -1,32767); END_IF		(* activate 'Message Hold Time' to avoid log clathering by repeated OpMsg entries *)
	xMsg36[69].Reset 	:= 	(iReset_Msg36[69] < 1);		//.Reset := TRUE;
	xMsg36[69]();
	MM2VIS.bMsg3669		:=	xMsg36[69].Q;

	xMsg36[70].Enable	:=	IN_CU.tPB2MM.bParaSetupOk ;
	xMsg36[70].Set		:=	OUT_CU.bMsg3670;(* B3670 reserve operating message *)
	IF xMsg36[70].Set THEN iReset_Msg36[70] := iDelay_MsgAutoReset_100ms; ELSE iReset_Msg36[70] := LIMIT(0, iReset_Msg36[70] -1,32767); END_IF		(* activate 'Message Hold Time' to avoid log clathering by repeated OpMsg entries *)
	xMsg36[70].Reset 	:= 	(iReset_Msg36[70] < 1);		//.Reset := TRUE;
	xMsg36[70]();
	MM2VIS.bMsg3670		:=	xMsg36[70].Q;
	(*----------------------------------------------------------------------*)

	xMsg36[71].Enable	:=	IN_CU.tPB2MM.bParaSetupOk ;
	xMsg36[71].Set		:=	OUT_CU.bMsg3671;(* B3671 reserve operating message *)
	IF xMsg36[71].Set THEN iReset_Msg36[71] := iDelay_MsgAutoReset_100ms; ELSE iReset_Msg36[71] := LIMIT(0, iReset_Msg36[71] -1,32767); END_IF		(* activate 'Message Hold Time' to avoid log clathering by repeated OpMsg entries *)
	xMsg36[71].Reset 	:= 	(iReset_Msg36[71] < 1);		//.Reset := TRUE;
	xMsg36[71]();
	MM2VIS.bMsg3671		:=	xMsg36[71].Q;

	xMsg36[72].Enable	:=	IN_CU.tPB2MM.bParaSetupOk ;
	xMsg36[72].Set		:=	OUT_CU.bMsg3672;(* B3672 reserve operating message *)
	IF xMsg36[72].Set THEN iReset_Msg36[72] := iDelay_MsgAutoReset_100ms; ELSE iReset_Msg36[72] := LIMIT(0, iReset_Msg36[72] -1,32767); END_IF		(* activate 'Message Hold Time' to avoid log clathering by repeated OpMsg entries *)
	xMsg36[72].Reset 	:= 	(iReset_Msg36[72] < 1);		//.Reset := TRUE;
	xMsg36[72]();
	MM2VIS.bMsg3672		:=	xMsg36[72].Q;
```
